   1:L PR[91] R[100]mm/sec CNT100;
   1:  PR[GP1:91,1] = PR[GP1:90,1] + -54.768;
   1:  PR[GP1:91,2] = PR[GP1:90,2] + 21.323;
   1:L PR[91] R[100]mm/sec CNT100;
   1:  PR[GP1:91,1] = PR[GP1:90,1] + -59.783;
   1:  PR[GP1:91,2] = PR[GP1:90,2] + 12.944;
   1:L PR[91] R[100]mm/sec CNT100;
   1:  PR[GP1:91,1] = PR[GP1:90,1] + -60.363;
   1:  PR[GP1:91,2] = PR[GP1:90,2] + 10.978;
   1:L PR[91] R[100]mm/sec CNT100;
   1:  PR[GP1:91,1] = PR[GP1:90,1] + -60.560;
   1:  PR[GP1:91,2] = PR[GP1:90,2] + 8.823;
   1:L PR[91] R[100]mm/sec CNT100;
   1:  PR[GP1:91,1] = PR[GP1:90,1] + -62.205;
   1:  PR[GP1:91,2] = PR[GP1:90,2] + -0.100;
   1:L PR[91] R[100]mm/sec CNT100;
   1:  PR[GP1:91,1] = PR[GP1:90,1] + -62.009;
   1:  PR[GP1:91,2] = PR[GP1:90,2] + -2.267;
   1:L PR[91] R[100]mm/sec CNT100;
   1:  PR[GP1:91,1] = PR[GP1:90,1] + -60.370;
   1:  PR[GP1:91,2] = PR[GP1:90,2] + -11.098;
   1:L PR[91] R[100]mm/sec CNT100;
   1:  PR[GP1:91,1] = PR[GP1:90,1] + -59.777;
   1:  PR[GP1:91,2] = PR[GP1:90,2] + -13.111;
   1:L PR[91] R[100]mm/sec CNT100;
   1:  PR[GP1:91,1] = PR[GP1:90,1] + -58.814;
   1:  PR[GP1:91,2] = PR[GP1:90,2] + -14.997;
   1:L PR[91] R[100]mm/sec CNT100;
   1:  PR[GP1:91,1] = PR[GP1:90,1] + -53.831;
   1:  PR[GP1:91,2] = PR[GP1:90,2] + -23.288;
   1:L PR[91] R[100]mm/sec CNT100;
   1:  PR[GP1:91,1] = PR[GP1:90,1] + -52.724;
   1:  PR[GP1:91,2] = PR[GP1:90,2] + -24.729;
   1:L PR[91] R[100]mm/sec CNT100;
   1:  PR[GP1:91,1] = PR[GP1:90,1] + -51.475;
   1:  PR[GP1:91,2] = PR[GP1:90,2] + -25.850;
   1:L PR[91] R[100]mm/sec CNT100;
   1:  PR[GP1:91,1] = PR[GP1:90,1] + -43.113;
   1:  PR[GP1:91,2] = PR[GP1:90,2] + -32.589;
   1:L PR[91] R[100]mm/sec CNT100;
   1:  PR[GP1:91,1] = PR[GP1:90,1] + -41.986;
   1:  PR[GP1:91,2] = PR[GP1:90,2] + -33.291;
   1:L PR[91] R[100]mm/sec CNT100;
   1:  PR[GP1:91,1] = PR[GP1:90,1] + -40.875;
   1:  PR[GP1:91,2] = PR[GP1:90,2] + -33.737;
   1:L PR[91] R[100]mm/sec CNT100;
   1:  PR[GP1:91,1] = PR[GP1:90,1] + -29.510;
   1:  PR[GP1:91,2] = PR[GP1:90,2] + -37.747;
   1:L PR[91] R[100]mm/sec CNT100;
   1:  PR[GP1:91,1] = PR[GP1:90,1] + -28.836;
   1:  PR[GP1:91,2] = PR[GP1:90,2] + -37.892;
   1:L PR[91] R[100]mm/sec CNT100;
   1:  PR[GP1:91,1] = PR[GP1:90,1] + -28.211;
   1:  PR[GP1:91,2] = PR[GP1:90,2] + -37.917;
   1:L PR[91] R[100]mm/sec CNT100;
   1:  PR[GP1:91,1] = PR[GP1:90,1] + -14.890;
   1:  PR[GP1:91,2] = PR[GP1:90,2] + -37.959;
   1:L PR[91] R[100]mm/sec CNT100;
   1:  PR[GP1:91,1] = PR[GP1:90,1] + -14.841;
   1:  PR[GP1:91,2] = PR[GP1:90,2] + -37.952;
   1:L PR[91] R[100]mm/sec CNT100;
   1:  PR[GP1:91,1] = PR[GP1:90,1] + -14.779;
   1:  PR[GP1:91,2] = PR[GP1:90,2] + -37.932;
   1:L PR[91] R[100]mm/sec CNT100;
   1:  PR[GP1:91,1] = PR[GP1:90,1] + -11.835;
   1:  PR[GP1:91,2] = PR[GP1:90,2] + -36.909;
   1:L PR[91] R[100]mm/sec CNT100;
   1:  PR[GP1:91,1] = PR[GP1:90,1] + -2.186;
   1:  PR[GP1:91,2] = PR[GP1:90,2] + -33.761;
   1:L PR[91] R[100]mm/sec CNT100;
   1:  PR[GP1:91,1] = PR[GP1:90,1] + -0.355;
   1:  PR[GP1:91,2] = PR[GP1:90,2] + -33.769;
   1:L PR[91] R[100]mm/sec CNT100;
   1:  PR[GP1:91,1] = PR[GP1:90,1] + 1.412;
   1:  PR[GP1:91,2] = PR[GP1:90,2] + -33.699;
   1:L PR[91] R[100]mm/sec CNT100;
   1:  PR[GP1:91,1] = PR[GP1:90,1] + 2.210;
   1:  PR[GP1:91,2] = PR[GP1:90,2] + -33.528;
   1:L PR[91] R[100]mm/sec CNT100;
   1:  PR[GP1:91,1] = PR[GP1:90,1] + 2.588;
   1:  PR[GP1:91,2] = PR[GP1:90,2] + -33.832;
   1:L PR[91] R[100]mm/sec CNT100;
   1:  PR[GP1:91,1] = PR[GP1:90,1] + 12.046;
   1:  PR[GP1:91,2] = PR[GP1:90,2] + -36.909;
   1:L PR[91] R[100]mm/sec CNT100;
   1:  PR[GP1:91,1] = PR[GP1:90,1] + 15.059;
   1:  PR[GP1:91,2] = PR[GP1:90,2] + -37.952;
   1:L PR[91] R[100]mm/sec CNT100;
   1:  PR[GP1:91,1] = PR[GP1:90,1] + 15.099;
   1:  PR[GP1:91,2] = PR[GP1:90,2] + -37.958;
   1:L PR[91] R[100]mm/sec CNT100;
   1:  PR[GP1:91,1] = PR[GP1:90,1] + 29.053;
   1:  PR[GP1:91,2] = PR[GP1:90,2] + -37.892;
   1:L PR[91] R[100]mm/sec CNT100;
   1:  PR[GP1:91,1] = PR[GP1:90,1] + 29.705;
   1:  PR[GP1:91,2] = PR[GP1:90,2] + -37.751;
   1:L PR[91] R[100]mm/sec CNT100;
   1:  PR[GP1:91,1] = PR[GP1:90,1] + 30.492;
   1:  PR[GP1:91,2] = PR[GP1:90,2] + -37.441;
   1:L PR[91] R[100]mm/sec CNT100;
   1:  PR[GP1:91,1] = PR[GP1:90,1] + 42.202;
   1:  PR[GP1:91,2] = PR[GP1:90,2] + -33.291;
   1:L PR[91] R[100]mm/sec CNT100;
   1:  PR[GP1:91,1] = PR[GP1:90,1] + 43.299;
   1:  PR[GP1:91,2] = PR[GP1:90,2] + -32.611;
   1:L PR[91] R[100]mm/sec CNT100;
   1:  PR[GP1:91,1] = PR[GP1:90,1] + 44.416;
   1:  PR[GP1:91,2] = PR[GP1:90,2] + -31.622;
   1:L PR[91] R[100]mm/sec CNT100;
   1:  PR[GP1:91,1] = PR[GP1:90,1] + 52.923;
   1:  PR[GP1:91,2] = PR[GP1:90,2] + -24.736;
   1:L PR[91] R[100]mm/sec CNT100;
   1:  PR[GP1:91,1] = PR[GP1:90,1] + 54.021;
   1:  PR[GP1:91,2] = PR[GP1:90,2] + -23.310;
   1:L PR[91] R[100]mm/sec CNT100;
   1:  PR[GP1:91,1] = PR[GP1:90,1] + 54.968;
   1:  PR[GP1:91,2] = PR[GP1:90,2] + -21.493;
   1:L PR[91] R[100]mm/sec CNT100;
   1:  PR[GP1:91,1] = PR[GP1:90,1] + 59.987;
   1:  PR[GP1:91,2] = PR[GP1:90,2] + -13.131;
   1:L PR[91] R[100]mm/sec CNT100;
   1:  PR[GP1:91,1] = PR[GP1:90,1] + 60.565;
   1:  PR[GP1:91,2] = PR[GP1:90,2] + -11.196;
   1:L PR[91] R[100]mm/sec CNT100;
   1:  PR[GP1:91,1] = PR[GP1:90,1] + 60.772;
   1:  PR[GP1:91,2] = PR[GP1:90,2] + -8.982;
   1:L PR[91] R[100]mm/sec CNT100;
   1:  PR[GP1:91,1] = PR[GP1:90,1] + 62.418;
   1:  PR[GP1:91,2] = PR[GP1:90,2] + -0.045;
   1:L PR[91] R[100]mm/sec CNT100;
   1:  PR[GP1:91,1] = PR[GP1:90,1] + 62.212;
   1:  PR[GP1:91,2] = PR[GP1:90,2] + 2.185;
   1:L PR[91] R[100]mm/sec CNT100;
   1:  PR[GP1:91,1] = PR[GP1:90,1] + 60.574;
   1:  PR[GP1:91,2] = PR[GP1:90,2] + 11.023;
   1:L PR[91] R[100]mm/sec CNT100;
   1:  PR[GP1:91,1] = PR[GP1:90,1] + 59.982;
   1:  PR[GP1:91,2] = PR[GP1:90,2] + 13.003;
   1:L PR[91] R[100]mm/sec CNT100;
   1:  PR[GP1:91,1] = PR[GP1:90,1] + 59.017;
   1:  PR[GP1:91,2] = PR[GP1:90,2] + 14.874;
   1:L PR[91] R[100]mm/sec CNT100;
   1:  PR[GP1:91,1] = PR[GP1:90,1] + 54.037;
   1:  PR[GP1:91,2] = PR[GP1:90,2] + 23.147;
   1:L PR[91] R[100]mm/sec CNT100;
   1:  PR[GP1:91,1] = PR[GP1:90,1] + 52.918;
   1:  PR[GP1:91,2] = PR[GP1:90,2] + 24.599;
   1:L PR[91] R[100]mm/sec CNT100;
   1:  PR[GP1:91,1] = PR[GP1:90,1] + 51.675;
   1:  PR[GP1:91,2] = PR[GP1:90,2] + 25.710;
   1:L PR[91] R[100]mm/sec CNT100;
   1:  PR[GP1:91,1] = PR[GP1:90,1] + 43.320;
   1:  PR[GP1:91,2] = PR[GP1:90,2] + 32.454;
   1:L PR[91] R[100]mm/sec CNT100;
   1:  PR[GP1:91,1] = PR[GP1:90,1] + 42.201;
   1:  PR[GP1:91,2] = PR[GP1:90,2] + 33.148;
   1:L PR[91] R[100]mm/sec CNT100;
   1:  PR[GP1:91,1] = PR[GP1:90,1] + 41.088;
   1:  PR[GP1:91,2] = PR[GP1:90,2] + 33.593;
   1:L PR[91] R[100]mm/sec CNT100;
   1:  PR[GP1:91,1] = PR[GP1:90,1] + 29.731;
   1:  PR[GP1:91,2] = PR[GP1:90,2] + 37.602;
   1:L PR[91] R[100]mm/sec CNT100;
   1:  PR[GP1:91,1] = PR[GP1:90,1] + 29.058;
   1:  PR[GP1:91,2] = PR[GP1:90,2] + 37.747;
   1:L PR[91] R[100]mm/sec CNT100;
   1:  PR[GP1:91,1] = PR[GP1:90,1] + 28.436;
   1:  PR[GP1:91,2] = PR[GP1:90,2] + 37.770;
   1:L PR[91] R[100]mm/sec CNT100;
   1:  PR[GP1:91,1] = PR[GP1:90,1] + 15.122;
   1:  PR[GP1:91,2] = PR[GP1:90,2] + 37.817;
   1:L PR[91] R[100]mm/sec CNT100;
   1:  PR[GP1:91,1] = PR[GP1:90,1] + 15.080;
   1:  PR[GP1:91,2] = PR[GP1:90,2] + 37.812;
   1:L PR[91] R[100]mm/sec CNT100;
   1:  PR[GP1:91,1] = PR[GP1:90,1] + 11.996;
   1:  PR[GP1:91,2] = PR[GP1:90,2] + 36.746;
   1:L PR[91] R[100]mm/sec CNT100;
   1:  PR[GP1:91,1] = PR[GP1:90,1] + 2.808;
   1:  PR[GP1:91,2] = PR[GP1:90,2] + 33.760;
   1:L PR[91] R[100]mm/sec CNT100;
   1:  PR[GP1:91,1] = PR[GP1:90,1] + 2.180;
   1:  PR[GP1:91,2] = PR[GP1:90,2] + 33.410;
   1:L PR[91] R[100]mm/sec CNT100;
   1:  ! -- Layer/Ebene 117 -- !;
   1:  PR[91] = PR[90];
   1:  PR[GP1:91,1] = PR[GP1:90,1] + 0.156;
   1:  PR[GP1:91,2] = PR[GP1:90,2] + 33.822;
   1:  PR[GP1:91,3] = PR[GP1:90,3] + 71.675;
   1:L PR[91] R[100]mm/sec CNT100;
   1:  PR[GP1:91,1] = PR[GP1:90,1] + -2.159;
   1:  PR[GP1:91,2] = PR[GP1:90,2] + 33.808;
   1:L PR[91] R[100]mm/sec CNT100;
   1:  PR[GP1:91,1] = PR[GP1:90,1] + -14.621;
   1:  PR[GP1:91,2] = PR[GP1:90,2] + 37.873;
   1:L PR[91] R[100]mm/sec CNT100;
   1:  PR[GP1:91,1] = PR[GP1:90,1] + -28.674;
   1:  PR[GP1:91,2] = PR[GP1:90,2] + 37.800;
   1:L PR[91] R[100]mm/sec CNT100;
   1:  PR[GP1:91,1] = PR[GP1:90,1] + -29.170;
   1:  PR[GP1:91,2] = PR[GP1:90,2] + 37.693;
   1:L PR[91] R[100]mm/sec CNT100;
   1:  PR[GP1:91,1] = PR[GP1:90,1] + -29.787;
   1:  PR[GP1:91,2] = PR[GP1:90,2] + 37.449;
   1:L PR[91] R[100]mm/sec CNT100;
   1:  PR[GP1:91,1] = PR[GP1:90,1] + -41.823;
   1:  PR[GP1:91,2] = PR[GP1:90,2] + 33.175;
   1:L PR[91] R[100]mm/sec CNT100;
   1:  PR[GP1:91,1] = PR[GP1:90,1] + -42.785;
   1:  PR[GP1:91,2] = PR[GP1:90,2] + 32.575;
   1:L PR[91] R[100]mm/sec CNT100;
   1:  PR[GP1:91,1] = PR[GP1:90,1] + -43.774;
   1:  PR[GP1:91,2] = PR[GP1:90,2] + 31.698;
   1:L PR[91] R[100]mm/sec CNT100;
   1:  PR[GP1:91,1] = PR[GP1:90,1] + -52.554;
   1:  PR[GP1:91,2] = PR[GP1:90,2] + 24.593;
   1:L PR[91] R[100]mm/sec CNT100;
   1:  PR[GP1:91,1] = PR[GP1:90,1] + -53.539;
   1:  PR[GP1:91,2] = PR[GP1:90,2] + 23.311;
   1:L PR[91] R[100]mm/sec CNT100;
   1:  PR[GP1:91,1] = PR[GP1:90,1] + -54.399;
   1:  PR[GP1:91,2] = PR[GP1:90,2] + 21.641;
   1:L PR[91] R[100]mm/sec CNT100;
   1:  PR[GP1:91,1] = PR[GP1:90,1] + -59.596;
   1:  PR[GP1:91,2] = PR[GP1:90,2] + 12.960;
   1:L PR[91] R[100]mm/sec CNT100;
   1:  PR[GP1:91,1] = PR[GP1:90,1] + -60.130;
   1:  PR[GP1:91,2] = PR[GP1:90,2] + 11.150;
   1:L PR[91] R[100]mm/sec CNT100;
   1:  PR[GP1:91,1] = PR[GP1:90,1] + -60.312;
   1:  PR[GP1:91,2] = PR[GP1:90,2] + 9.158;
   1:L PR[91] R[100]mm/sec CNT100;
   1:  PR[GP1:91,1] = PR[GP1:90,1] + -62.019;
   1:  PR[GP1:91,2] = PR[GP1:90,2] + -0.100;
   1:L PR[91] R[100]mm/sec CNT100;
   1:  PR[GP1:91,1] = PR[GP1:90,1] + -61.837;
   1:  PR[GP1:91,2] = PR[GP1:90,2] + -2.111;
   1:L PR[91] R[100]mm/sec CNT100;
   1:  PR[GP1:91,1] = PR[GP1:90,1] + -60.137;
   1:  PR[GP1:91,2] = PR[GP1:90,2] + -11.270;
   1:L PR[91] R[100]mm/sec CNT100;
   1:  PR[GP1:91,1] = PR[GP1:90,1] + -59.589;
   1:  PR[GP1:91,2] = PR[GP1:90,2] + -13.126;
   1:L PR[91] R[100]mm/sec CNT100;
   1:  PR[GP1:91,1] = PR[GP1:90,1] + -58.701;
   1:  PR[GP1:91,2] = PR[GP1:90,2] + -14.867;
   1:L PR[91] R[100]mm/sec CNT100;
   1:  PR[GP1:91,1] = PR[GP1:90,1] + -53.546;
   1:  PR[GP1:91,2] = PR[GP1:90,2] + -23.444;
   1:L PR[91] R[100]mm/sec CNT100;
   1:  PR[GP1:91,1] = PR[GP1:90,1] + -52.540;
   1:  PR[GP1:91,2] = PR[GP1:90,2] + -24.754;
   1:L PR[91] R[100]mm/sec CNT100;
   1:  PR[GP1:91,1] = PR[GP1:90,1] + -51.405;
   1:  PR[GP1:91,2] = PR[GP1:90,2] + -25.772;
   1:L PR[91] R[100]mm/sec CNT100;
   1:  PR[GP1:91,1] = PR[GP1:90,1] + -42.788;
   1:  PR[GP1:91,2] = PR[GP1:90,2] + -32.718;
   1:L PR[91] R[100]mm/sec CNT100;
   1:  PR[GP1:91,1] = PR[GP1:90,1] + -41.802;
   1:  PR[GP1:91,2] = PR[GP1:90,2] + -33.331;
   1:L PR[91] R[100]mm/sec CNT100;
   1:  PR[GP1:91,1] = PR[GP1:90,1] + -40.829;
   1:  PR[GP1:91,2] = PR[GP1:90,2] + -33.722;
   1:L PR[91] R[100]mm/sec CNT100;
   1:  PR[GP1:91,1] = PR[GP1:90,1] + -29.164;
   1:  PR[GP1:91,2] = PR[GP1:90,2] + -37.838;
   1:L PR[91] R[100]mm/sec CNT100;
   1:  PR[GP1:91,1] = PR[GP1:90,1] + -28.648;
   1:  PR[GP1:91,2] = PR[GP1:90,2] + -37.949;
   1:L PR[91] R[100]mm/sec CNT100;
   1:  PR[GP1:91,1] = PR[GP1:90,1] + -28.166;
   1:  PR[GP1:91,2] = PR[GP1:90,2] + -37.968;
   1:L PR[91] R[100]mm/sec CNT100;
   1:  PR[GP1:91,1] = PR[GP1:90,1] + -14.623;
   1:  PR[GP1:91,2] = PR[GP1:90,2] + -38.014;
   1:L PR[91] R[100]mm/sec CNT100;
   1:  PR[GP1:91,1] = PR[GP1:90,1] + -2.159;
   1:  PR[GP1:91,2] = PR[GP1:90,2] + -33.955;
   1:L PR[91] R[100]mm/sec CNT100;
   1:  PR[GP1:91,1] = PR[GP1:90,1] + 0.246;
   1:  PR[GP1:91,2] = PR[GP1:90,2] + -33.967;
   1:L PR[91] R[100]mm/sec CNT100;
   1:  PR[GP1:91,1] = PR[GP1:90,1] + 1.578;
   1:  PR[GP1:91,2] = PR[GP1:90,2] + -33.913;
   1:L PR[91] R[100]mm/sec CNT100;
   1:  PR[GP1:91,1] = PR[GP1:90,1] + 2.241;
   1:  PR[GP1:91,2] = PR[GP1:90,2] + -33.772;
   1:L PR[91] R[100]mm/sec CNT100;
   1:  PR[GP1:91,1] = PR[GP1:90,1] + 2.561;
   1:  PR[GP1:91,2] = PR[GP1:90,2] + -34.030;
   1:L PR[91] R[100]mm/sec CNT100;
   1:  PR[GP1:91,1] = PR[GP1:90,1] + 14.808;
   1:  PR[GP1:91,2] = PR[GP1:90,2] + -38.012;
   1:L PR[91] R[100]mm/sec CNT100;
   1:  PR[GP1:91,1] = PR[GP1:90,1] + 28.865;
   1:  PR[GP1:91,2] = PR[GP1:90,2] + -37.948;
   1:L PR[91] R[100]mm/sec CNT100;
   1:  PR[GP1:91,1] = PR[GP1:90,1] + 29.360;
   1:  PR[GP1:91,2] = PR[GP1:90,2] + -37.842;
   1:L PR[91] R[100]mm/sec CNT100;
   1:  PR[GP1:91,1] = PR[GP1:90,1] + 29.977;
   1:  PR[GP1:91,2] = PR[GP1:90,2] + -37.599;
   1:L PR[91] R[100]mm/sec CNT100;
   1:  PR[GP1:91,1] = PR[GP1:90,1] + 42.019;
   1:  PR[GP1:91,2] = PR[GP1:90,2] + -33.331;
   1:L PR[91] R[100]mm/sec CNT100;
   1:  PR[GP1:91,1] = PR[GP1:90,1] + 42.976;
   1:  PR[GP1:91,2] = PR[GP1:90,2] + -32.738;
   1:L PR[91] R[100]mm/sec CNT100;
   1:  PR[GP1:91,1] = PR[GP1:90,1] + 43.957;
   1:  PR[GP1:91,2] = PR[GP1:90,2] + -31.869;
   1:L PR[91] R[100]mm/sec CNT100;
   1:  PR[GP1:91,1] = PR[GP1:90,1] + 52.741;
   1:  PR[GP1:91,2] = PR[GP1:90,2] + -24.758;
   1:L PR[91] R[100]mm/sec CNT100;
   1:  PR[GP1:91,1] = PR[GP1:90,1] + 53.737;
   1:  PR[GP1:91,2] = PR[GP1:90,2] + -23.465;
   1:L PR[91] R[100]mm/sec CNT100;
   1:  PR[GP1:91,1] = PR[GP1:90,1] + 54.600;
   1:  PR[GP1:91,2] = PR[GP1:90,2] + -21.809;
   1:L PR[91] R[100]mm/sec CNT100;
   1:  PR[GP1:91,1] = PR[GP1:90,1] + 59.801;
   1:  PR[GP1:91,2] = PR[GP1:90,2] + -13.145;
   1:L PR[91] R[100]mm/sec CNT100;
   1:  PR[GP1:91,1] = PR[GP1:90,1] + 60.333;
   1:  PR[GP1:91,2] = PR[GP1:90,2] + -11.363;
   1:L PR[91] R[100]mm/sec CNT100;
   1:  PR[GP1:91,1] = PR[GP1:90,1] + 60.524;
   1:  PR[GP1:91,2] = PR[GP1:90,2] + -9.317;
   1:L PR[91] R[100]mm/sec CNT100;
   1:  PR[GP1:91,1] = PR[GP1:90,1] + 62.232;
   1:  PR[GP1:91,2] = PR[GP1:90,2] + -0.045;
   1:L PR[91] R[100]mm/sec CNT100;
   1:  PR[GP1:91,1] = PR[GP1:90,1] + 62.041;
   1:  PR[GP1:91,2] = PR[GP1:90,2] + 2.024;
   1:L PR[91] R[100]mm/sec CNT100;
   1:  PR[GP1:91,1] = PR[GP1:90,1] + 60.342;
   1:  PR[GP1:91,2] = PR[GP1:90,2] + 11.191;
   1:L PR[91] R[100]mm/sec CNT100;
   1:  PR[GP1:91,1] = PR[GP1:90,1] + 59.796;
   1:  PR[GP1:91,2] = PR[GP1:90,2] + 13.017;
   1:L PR[91] R[100]mm/sec CNT100;
   1:  PR[GP1:91,1] = PR[GP1:90,1] + 58.905;
   1:  PR[GP1:91,2] = PR[GP1:90,2] + 14.743;
   1:L PR[91] R[100]mm/sec CNT100;
   1:  PR[GP1:91,1] = PR[GP1:90,1] + 53.753;
   1:  PR[GP1:91,2] = PR[GP1:90,2] + 23.301;
   1:L PR[91] R[100]mm/sec CNT100;
   1:  PR[GP1:91,1] = PR[GP1:90,1] + 52.737;
   1:  PR[GP1:91,2] = PR[GP1:90,2] + 24.621;
   1:L PR[91] R[100]mm/sec CNT100;
   1:  PR[GP1:91,1] = PR[GP1:90,1] + 51.607;
   1:  PR[GP1:91,2] = PR[GP1:90,2] + 25.631;
   1:L PR[91] R[100]mm/sec CNT100;
   1:  PR[GP1:91,1] = PR[GP1:90,1] + 42.997;
   1:  PR[GP1:91,2] = PR[GP1:90,2] + 32.581;
   1:L PR[91] R[100]mm/sec CNT100;
   1:  PR[GP1:91,1] = PR[GP1:90,1] + 42.019;
   1:  PR[GP1:91,2] = PR[GP1:90,2] + 33.188;
   1:L PR[91] R[100]mm/sec CNT100;
   1:  PR[GP1:91,1] = PR[GP1:90,1] + 41.044;
   1:  PR[GP1:91,2] = PR[GP1:90,2] + 33.577;
   1:L PR[91] R[100]mm/sec CNT100;
   1:  PR[GP1:91,1] = PR[GP1:90,1] + 29.387;
   1:  PR[GP1:91,2] = PR[GP1:90,2] + 37.693;
   1:L PR[91] R[100]mm/sec CNT100;
   1:  PR[GP1:91,1] = PR[GP1:90,1] + 28.871;
   1:  PR[GP1:91,2] = PR[GP1:90,2] + 37.803;
   1:L PR[91] R[100]mm/sec CNT100;
   1:  PR[GP1:91,1] = PR[GP1:90,1] + 28.391;
   1:  PR[GP1:91,2] = PR[GP1:90,2] + 37.822;
   1:L PR[91] R[100]mm/sec CNT100;
   1:  PR[GP1:91,1] = PR[GP1:90,1] + 14.829;
   1:  PR[GP1:91,2] = PR[GP1:90,2] + 37.872;
   1:L PR[91] R[100]mm/sec CNT100;
   1:  PR[GP1:91,1] = PR[GP1:90,1] + 2.720;
   1:  PR[GP1:91,2] = PR[GP1:90,2] + 33.937;
   1:L PR[91] R[100]mm/sec CNT100;
   1:  PR[GP1:91,1] = PR[GP1:90,1] + 2.210;
   1:  PR[GP1:91,2] = PR[GP1:90,2] + 33.653;
   1:L PR[91] R[100]mm/sec CNT100;
   1:  ! -- Layer/Ebene 118 -- !;
   1:  PR[91] = PR[90];
   1:  PR[GP1:91,1] = PR[GP1:90,1] + 0.747;
   1:  PR[GP1:91,2] = PR[GP1:90,2] + 34.019;
   1:  PR[GP1:91,3] = PR[GP1:90,3] + 72.285;
   1:L PR[91] R[100]mm/sec CNT100;
   1:  PR[GP1:91,1] = PR[GP1:90,1] + -2.132;
   1:  PR[GP1:91,2] = PR[GP1:90,2] + 34.002;
   1:L PR[91] R[100]mm/sec CNT100;
   1:  PR[GP1:91,1] = PR[GP1:90,1] + -13.373;
   1:  PR[GP1:91,2] = PR[GP1:90,2] + 37.669;
   1:L PR[91] R[100]mm/sec CNT100;
   1:  PR[GP1:91,1] = PR[GP1:90,1] + -14.331;
   1:  PR[GP1:91,2] = PR[GP1:90,2] + 37.965;
   1:L PR[91] R[100]mm/sec CNT100;
   1:  PR[GP1:91,1] = PR[GP1:90,1] + -14.593;
   1:  PR[GP1:91,2] = PR[GP1:90,2] + 37.974;
   1:L PR[91] R[100]mm/sec CNT100;
   1:  PR[GP1:91,1] = PR[GP1:90,1] + -18.226;
   1:  PR[GP1:91,2] = PR[GP1:90,2] + 37.908;
   1:L PR[91] R[100]mm/sec CNT100;
   1:  PR[GP1:91,1] = PR[GP1:90,1] + -28.487;
   1:  PR[GP1:91,2] = PR[GP1:90,2] + 37.857;
   1:L PR[91] R[100]mm/sec CNT100;
   1:  PR[GP1:91,1] = PR[GP1:90,1] + -28.825;
   1:  PR[GP1:91,2] = PR[GP1:90,2] + 37.784;
   1:L PR[91] R[100]mm/sec CNT100;
   1:  PR[GP1:91,1] = PR[GP1:90,1] + -29.271;
   1:  PR[GP1:91,2] = PR[GP1:90,2] + 37.607;
   1:L PR[91] R[100]mm/sec CNT100;
   1:  PR[GP1:91,1] = PR[GP1:90,1] + -41.639;
   1:  PR[GP1:91,2] = PR[GP1:90,2] + 33.215;
   1:L PR[91] R[100]mm/sec CNT100;
   1:  PR[GP1:91,1] = PR[GP1:90,1] + -42.461;
   1:  PR[GP1:91,2] = PR[GP1:90,2] + 32.704;
   1:L PR[91] R[100]mm/sec CNT100;
   1:  PR[GP1:91,1] = PR[GP1:90,1] + -43.313;
   1:  PR[GP1:91,2] = PR[GP1:90,2] + 31.946;
   1:L PR[91] R[100]mm/sec CNT100;
   1:  PR[GP1:91,1] = PR[GP1:90,1] + -52.371;
   1:  PR[GP1:91,2] = PR[GP1:90,2] + 24.617;
   1:L PR[91] R[100]mm/sec CNT100;
   1:  PR[GP1:91,1] = PR[GP1:90,1] + -53.254;
   1:  PR[GP1:91,2] = PR[GP1:90,2] + 23.467;
   1:L PR[91] R[100]mm/sec CNT100;
   1:  PR[GP1:91,1] = PR[GP1:90,1] + -54.031;
   1:  PR[GP1:91,2] = PR[GP1:90,2] + 21.959;
   1:L PR[91] R[100]mm/sec CNT100;
   1:  PR[GP1:91,1] = PR[GP1:90,1] + -59.409;
   1:  PR[GP1:91,2] = PR[GP1:90,2] + 12.975;
   1:L PR[91] R[100]mm/sec CNT100;
   1:  PR[GP1:91,1] = PR[GP1:90,1] + -59.897;
   1:  PR[GP1:91,2] = PR[GP1:90,2] + 11.321;
   1:L PR[91] R[100]mm/sec CNT100;
   1:  PR[GP1:91,1] = PR[GP1:90,1] + -60.064;
   1:  PR[GP1:91,2] = PR[GP1:90,2] + 9.492;
   1:L PR[91] R[100]mm/sec CNT100;
   1:  PR[GP1:91,1] = PR[GP1:90,1] + -61.832;
   1:  PR[GP1:91,2] = PR[GP1:90,2] + -0.100;
   1:L PR[91] R[100]mm/sec CNT100;
   1:  PR[GP1:91,1] = PR[GP1:90,1] + -61.665;
   1:  PR[GP1:91,2] = PR[GP1:90,2] + -1.954;
   1:L PR[91] R[100]mm/sec CNT100;
   1:  PR[GP1:91,1] = PR[GP1:90,1] + -59.903;
   1:  PR[GP1:91,2] = PR[GP1:90,2] + -11.442;
   1:L PR[91] R[100]mm/sec CNT100;
   1:  PR[GP1:91,1] = PR[GP1:90,1] + -59.402;
   1:  PR[GP1:91,2] = PR[GP1:90,2] + -13.142;
   1:L PR[91] R[100]mm/sec CNT100;
   1:  PR[GP1:91,1] = PR[GP1:90,1] + -58.589;
   1:  PR[GP1:91,2] = PR[GP1:90,2] + -14.737;
   1:L PR[91] R[100]mm/sec CNT100;
   1:  PR[GP1:91,1] = PR[GP1:90,1] + -53.262;
   1:  PR[GP1:91,2] = PR[GP1:90,2] + -23.600;
   1:L PR[91] R[100]mm/sec CNT100;
   1:  PR[GP1:91,1] = PR[GP1:90,1] + -52.357;
   1:  PR[GP1:91,2] = PR[GP1:90,2] + -24.778;
   1:L PR[91] R[100]mm/sec CNT100;
   1:  PR[GP1:91,1] = PR[GP1:90,1] + -51.334;
   1:  PR[GP1:91,2] = PR[GP1:90,2] + -25.695;
   1:L PR[91] R[100]mm/sec CNT100;
   1:  PR[GP1:91,1] = PR[GP1:90,1] + -42.462;
   1:  PR[GP1:91,2] = PR[GP1:90,2] + -32.846;
   1:L PR[91] R[100]mm/sec CNT100;
   1:  PR[GP1:91,1] = PR[GP1:90,1] + -41.619;
   1:  PR[GP1:91,2] = PR[GP1:90,2] + -33.371;
   1:L PR[91] R[100]mm/sec CNT100;
   1:  PR[GP1:91,1] = PR[GP1:90,1] + -40.783;
   1:  PR[GP1:91,2] = PR[GP1:90,2] + -33.707;
   1:L PR[91] R[100]mm/sec CNT100;
   1:  PR[GP1:91,1] = PR[GP1:90,1] + -28.818;
   1:  PR[GP1:91,2] = PR[GP1:90,2] + -37.928;
   1:L PR[91] R[100]mm/sec CNT100;
   1:  PR[GP1:91,1] = PR[GP1:90,1] + -28.460;
   1:  PR[GP1:91,2] = PR[GP1:90,2] + -38.006;
   1:L PR[91] R[100]mm/sec CNT100;
   1:  PR[GP1:91,1] = PR[GP1:90,1] + -28.120;
   1:  PR[GP1:91,2] = PR[GP1:90,2] + -38.019;
   1:L PR[91] R[100]mm/sec CNT100;
   1:  PR[GP1:91,1] = PR[GP1:90,1] + -18.226;
   1:  PR[GP1:91,2] = PR[GP1:90,2] + -38.050;
   1:L PR[91] R[100]mm/sec CNT100;
   1:  PR[GP1:91,1] = PR[GP1:90,1] + -14.573;
   1:  PR[GP1:91,2] = PR[GP1:90,2] + -38.115;
   1:L PR[91] R[100]mm/sec CNT100;
   1:  PR[GP1:91,1] = PR[GP1:90,1] + -14.309;
   1:  PR[GP1:91,2] = PR[GP1:90,2] + -38.106;
   1:L PR[91] R[100]mm/sec CNT100;
   1:  PR[GP1:91,1] = PR[GP1:90,1] + -13.125;
   1:  PR[GP1:91,2] = PR[GP1:90,2] + -37.737;
   1:L PR[91] R[100]mm/sec CNT100;
   1:  PR[GP1:91,1] = PR[GP1:90,1] + -2.132;
   1:  PR[GP1:91,2] = PR[GP1:90,2] + -34.149;
   1:L PR[91] R[100]mm/sec CNT100;
   1:  PR[GP1:91,1] = PR[GP1:90,1] + 0.848;
   1:  PR[GP1:91,2] = PR[GP1:90,2] + -34.164;
   1:L PR[91] R[100]mm/sec CNT100;
   1:  PR[GP1:91,1] = PR[GP1:90,1] + 1.743;
   1:  PR[GP1:91,2] = PR[GP1:90,2] + -34.128;
   1:L PR[91] R[100]mm/sec CNT100;
   1:  PR[GP1:91,1] = PR[GP1:90,1] + 2.271;
   1:  PR[GP1:91,2] = PR[GP1:90,2] + -34.016;
   1:L PR[91] R[100]mm/sec CNT100;
   1:  PR[GP1:91,1] = PR[GP1:90,1] + 2.534;
   1:  PR[GP1:91,2] = PR[GP1:90,2] + -34.227;
   1:L PR[91] R[100]mm/sec CNT100;
   1:  PR[GP1:91,1] = PR[GP1:90,1] + 10.808;
   1:  PR[GP1:91,2] = PR[GP1:90,2] + -36.919;
   1:L PR[91] R[100]mm/sec CNT100;
   1:  PR[GP1:91,1] = PR[GP1:90,1] + 14.521;
   1:  PR[GP1:91,2] = PR[GP1:90,2] + -38.105;
   1:L PR[91] R[100]mm/sec CNT100;
   1:  PR[GP1:91,1] = PR[GP1:90,1] + 14.783;
   1:  PR[GP1:91,2] = PR[GP1:90,2] + -38.114;
   1:L PR[91] R[100]mm/sec CNT100;
   1:  PR[GP1:91,1] = PR[GP1:90,1] + 18.439;
   1:  PR[GP1:91,2] = PR[GP1:90,2] + -38.050;
   1:L PR[91] R[100]mm/sec CNT100;
   1:  PR[GP1:91,1] = PR[GP1:90,1] + 28.678;
   1:  PR[GP1:91,2] = PR[GP1:90,2] + -38.005;
   1:L PR[91] R[100]mm/sec CNT100;
   1:  PR[GP1:91,1] = PR[GP1:90,1] + 29.015;
   1:  PR[GP1:91,2] = PR[GP1:90,2] + -37.932;
   1:L PR[91] R[100]mm/sec CNT100;
   1:  PR[GP1:91,1] = PR[GP1:90,1] + 29.461;
   1:  PR[GP1:91,2] = PR[GP1:90,2] + -37.756;
   1:L PR[91] R[100]mm/sec CNT100;
   1:  PR[GP1:91,1] = PR[GP1:90,1] + 41.836;
   1:  PR[GP1:91,2] = PR[GP1:90,2] + -33.370;
   1:L PR[91] R[100]mm/sec CNT100;
   1:  PR[GP1:91,1] = PR[GP1:90,1] + 42.652;
   1:  PR[GP1:91,2] = PR[GP1:90,2] + -32.865;
   1:L PR[91] R[100]mm/sec CNT100;
   1:  PR[GP1:91,1] = PR[GP1:90,1] + 43.499;
   1:  PR[GP1:91,2] = PR[GP1:90,2] + -32.115;
   1:L PR[91] R[100]mm/sec CNT100;
   1:  PR[GP1:91,1] = PR[GP1:90,1] + 52.560;
   1:  PR[GP1:91,2] = PR[GP1:90,2] + -24.780;
   1:L PR[91] R[100]mm/sec CNT100;
   1:  PR[GP1:91,1] = PR[GP1:90,1] + 53.454;
   1:  PR[GP1:91,2] = PR[GP1:90,2] + -23.620;
   1:L PR[91] R[100]mm/sec CNT100;
   1:  PR[GP1:91,1] = PR[GP1:90,1] + 54.233;
   1:  PR[GP1:91,2] = PR[GP1:90,2] + -22.125;
   1:L PR[91] R[100]mm/sec CNT100;
   1:  PR[GP1:91,1] = PR[GP1:90,1] + 59.614;
   1:  PR[GP1:91,2] = PR[GP1:90,2] + -13.159;
   1:L PR[91] R[100]mm/sec CNT100;
   1:  PR[GP1:91,1] = PR[GP1:90,1] + 60.101;
   1:  PR[GP1:91,2] = PR[GP1:90,2] + -11.531;
   1:L PR[91] R[100]mm/sec CNT100;
   1:  PR[GP1:91,1] = PR[GP1:90,1] + 60.276;
   1:  PR[GP1:91,2] = PR[GP1:90,2] + -9.651;
   1:L PR[91] R[100]mm/sec CNT100;
   1:  PR[GP1:91,1] = PR[GP1:90,1] + 62.045;
   1:  PR[GP1:91,2] = PR[GP1:90,2] + -0.045;
   1:L PR[91] R[100]mm/sec CNT100;
   1:  PR[GP1:91,1] = PR[GP1:90,1] + 61.869;
   1:  PR[GP1:91,2] = PR[GP1:90,2] + 1.863;
   1:L PR[91] R[100]mm/sec CNT100;
   1:  PR[GP1:91,1] = PR[GP1:90,1] + 60.109;
   1:  PR[GP1:91,2] = PR[GP1:90,2] + 11.358;
   1:L PR[91] R[100]mm/sec CNT100;
   1:  PR[GP1:91,1] = PR[GP1:90,1] + 59.610;
   1:  PR[GP1:91,2] = PR[GP1:90,2] + 13.031;
   1:L PR[91] R[100]mm/sec CNT100;
   1:  PR[GP1:91,1] = PR[GP1:90,1] + 58.793;
   1:  PR[GP1:91,2] = PR[GP1:90,2] + 14.613;
   1:L PR[91] R[100]mm/sec CNT100;
   1:  PR[GP1:91,1] = PR[GP1:90,1] + 53.469;
   1:  PR[GP1:91,2] = PR[GP1:90,2] + 23.456;
   1:L PR[91] R[100]mm/sec CNT100;
   1:  PR[GP1:91,1] = PR[GP1:90,1] + 52.555;
   1:  PR[GP1:91,2] = PR[GP1:90,2] + 24.643;
   1:L PR[91] R[100]mm/sec CNT100;
   1:  PR[GP1:91,1] = PR[GP1:90,1] + 51.538;
   1:  PR[GP1:91,2] = PR[GP1:90,2] + 25.552;
   1:L PR[91] R[100]mm/sec CNT100;
   1:  PR[GP1:91,1] = PR[GP1:90,1] + 42.674;
   1:  PR[GP1:91,2] = PR[GP1:90,2] + 32.708;
   1:L PR[91] R[100]mm/sec CNT100;
   1:  PR[GP1:91,1] = PR[GP1:90,1] + 41.836;
   1:  PR[GP1:91,2] = PR[GP1:90,2] + 33.227;
   1:L PR[91] R[100]mm/sec CNT100;
   1:  PR[GP1:91,1] = PR[GP1:90,1] + 40.999;
   1:  PR[GP1:91,2] = PR[GP1:90,2] + 33.562;
   1:L PR[91] R[100]mm/sec CNT100;
   1:  PR[GP1:91,1] = PR[GP1:90,1] + 29.042;
   1:  PR[GP1:91,2] = PR[GP1:90,2] + 37.783;
   1:L PR[91] R[100]mm/sec CNT100;
   1:  PR[GP1:91,1] = PR[GP1:90,1] + 28.685;
   1:  PR[GP1:91,2] = PR[GP1:90,2] + 37.860;
   1:L PR[91] R[100]mm/sec CNT100;
   1:  PR[GP1:91,1] = PR[GP1:90,1] + 28.346;
   1:  PR[GP1:91,2] = PR[GP1:90,2] + 37.873;
   1:L PR[91] R[100]mm/sec CNT100;
   1:  PR[GP1:91,1] = PR[GP1:90,1] + 18.439;
   1:  PR[GP1:91,2] = PR[GP1:90,2] + 37.907;
   1:L PR[91] R[100]mm/sec CNT100;
   1:  PR[GP1:91,1] = PR[GP1:90,1] + 14.803;
   1:  PR[GP1:91,2] = PR[GP1:90,2] + 37.973;
   1:L PR[91] R[100]mm/sec CNT100;
   1:  PR[GP1:91,1] = PR[GP1:90,1] + 14.542;
   1:  PR[GP1:91,2] = PR[GP1:90,2] + 37.964;
   1:L PR[91] R[100]mm/sec CNT100;
   1:  PR[GP1:91,1] = PR[GP1:90,1] + 11.048;
   1:  PR[GP1:91,2] = PR[GP1:90,2] + 36.850;
   1:L PR[91] R[100]mm/sec CNT100;
   1:  PR[GP1:91,1] = PR[GP1:90,1] + 2.631;
   1:  PR[GP1:91,2] = PR[GP1:90,2] + 34.114;
   1:L PR[91] R[100]mm/sec CNT100;
   1:  PR[GP1:91,1] = PR[GP1:90,1] + 2.240;
   1:  PR[GP1:91,2] = PR[GP1:90,2] + 33.897;
   1:L PR[91] R[100]mm/sec CNT100;
   1:  ! -- Layer/Ebene 119 -- !;
   1:  PR[91] = PR[90];
   1:  PR[GP1:91,1] = PR[GP1:90,1] + 1.338;
   1:  PR[GP1:91,2] = PR[GP1:90,2] + 34.217;
   1:  PR[GP1:91,3] = PR[GP1:90,3] + 72.895;
   1:L PR[91] R[100]mm/sec CNT100;
   1:  PR[GP1:91,1] = PR[GP1:90,1] + -2.105;
   1:  PR[GP1:91,2] = PR[GP1:90,2] + 34.195;
   1:L PR[91] R[100]mm/sec CNT100;
   1:  PR[GP1:91,1] = PR[GP1:90,1] + -12.103;
   1:  PR[GP1:91,2] = PR[GP1:90,2] + 37.457;
   1:L PR[91] R[100]mm/sec CNT100;
   1:  PR[GP1:91,1] = PR[GP1:90,1] + -14.033;
   1:  PR[GP1:91,2] = PR[GP1:90,2] + 38.054;
   1:L PR[91] R[100]mm/sec CNT100;
   1:  PR[GP1:91,1] = PR[GP1:90,1] + -14.631;
   1:  PR[GP1:91,2] = PR[GP1:90,2] + 38.075;
   1:L PR[91] R[100]mm/sec CNT100;
   1:  PR[GP1:91,1] = PR[GP1:90,1] + -21.679;
   1:  PR[GP1:91,2] = PR[GP1:90,2] + 37.946;
   1:L PR[91] R[100]mm/sec CNT100;
   1:  PR[GP1:91,1] = PR[GP1:90,1] + -28.299;
   1:  PR[GP1:91,2] = PR[GP1:90,2] + 37.913;
   1:L PR[91] R[100]mm/sec CNT100;
   1:  PR[GP1:91,1] = PR[GP1:90,1] + -28.479;
   1:  PR[GP1:91,2] = PR[GP1:90,2] + 37.874;
   1:L PR[91] R[100]mm/sec CNT100;
   1:  PR[GP1:91,1] = PR[GP1:90,1] + -28.755;
   1:  PR[GP1:91,2] = PR[GP1:90,2] + 37.765;
   1:L PR[91] R[100]mm/sec CNT100;
   1:  PR[GP1:91,1] = PR[GP1:90,1] + -41.456;
   1:  PR[GP1:91,2] = PR[GP1:90,2] + 33.255;
   1:L PR[91] R[100]mm/sec CNT100;
   1:  PR[GP1:91,1] = PR[GP1:90,1] + -42.136;
   1:  PR[GP1:91,2] = PR[GP1:90,2] + 32.832;
   1:L PR[91] R[100]mm/sec CNT100;
   1:  PR[GP1:91,1] = PR[GP1:90,1] + -42.853;
   1:  PR[GP1:91,2] = PR[GP1:90,2] + 32.195;
   1:L PR[91] R[100]mm/sec CNT100;
   1:  PR[GP1:91,1] = PR[GP1:90,1] + -52.187;
   1:  PR[GP1:91,2] = PR[GP1:90,2] + 24.641;
   1:L PR[91] R[100]mm/sec CNT100;
   1:  PR[GP1:91,1] = PR[GP1:90,1] + -52.970;
   1:  PR[GP1:91,2] = PR[GP1:90,2] + 23.623;
   1:L PR[91] R[100]mm/sec CNT100;
   1:  PR[GP1:91,1] = PR[GP1:90,1] + -53.663;
   1:  PR[GP1:91,2] = PR[GP1:90,2] + 22.277;
   1:L PR[91] R[100]mm/sec CNT100;
   1:  PR[GP1:91,1] = PR[GP1:90,1] + -59.222;
   1:  PR[GP1:91,2] = PR[GP1:90,2] + 12.991;
   1:L PR[91] R[100]mm/sec CNT100;
   1:  PR[GP1:91,1] = PR[GP1:90,1] + -59.664;
   1:  PR[GP1:91,2] = PR[GP1:90,2] + 11.493;
   1:L PR[91] R[100]mm/sec CNT100;
   1:  PR[GP1:91,1] = PR[GP1:90,1] + -59.816;
   1:  PR[GP1:91,2] = PR[GP1:90,2] + 9.826;
   1:L PR[91] R[100]mm/sec CNT100;
   1:  PR[GP1:91,1] = PR[GP1:90,1] + -61.646;
   1:  PR[GP1:91,2] = PR[GP1:90,2] + -0.100;
   1:L PR[91] R[100]mm/sec CNT100;
   1:  PR[GP1:91,1] = PR[GP1:90,1] + -61.493;
   1:  PR[GP1:91,2] = PR[GP1:90,2] + -1.798;
   1:L PR[91] R[100]mm/sec CNT100;
   1:  PR[GP1:91,1] = PR[GP1:90,1] + -59.670;
   1:  PR[GP1:91,2] = PR[GP1:90,2] + -11.613;
   1:L PR[91] R[100]mm/sec CNT100;
   1:  PR[GP1:91,1] = PR[GP1:90,1] + -59.215;
   1:  PR[GP1:91,2] = PR[GP1:90,2] + -13.158;
   1:L PR[91] R[100]mm/sec CNT100;
   1:  PR[GP1:91,1] = PR[GP1:90,1] + -58.476;
   1:  PR[GP1:91,2] = PR[GP1:90,2] + -14.608;
   1:L PR[91] R[100]mm/sec CNT100;
   1:  PR[GP1:91,1] = PR[GP1:90,1] + -52.977;
   1:  PR[GP1:91,2] = PR[GP1:90,2] + -23.756;
   1:L PR[91] R[100]mm/sec CNT100;
   1:  PR[GP1:91,1] = PR[GP1:90,1] + -52.173;
   1:  PR[GP1:91,2] = PR[GP1:90,2] + -24.803;
   1:L PR[91] R[100]mm/sec CNT100;
   1:  PR[GP1:91,1] = PR[GP1:90,1] + -51.264;
   1:  PR[GP1:91,2] = PR[GP1:90,2] + -25.618;
   1:L PR[91] R[100]mm/sec CNT100;
   1:  PR[GP1:91,1] = PR[GP1:90,1] + -42.137;
   1:  PR[GP1:91,2] = PR[GP1:90,2] + -32.974;
   1:L PR[91] R[100]mm/sec CNT100;
   1:  PR[GP1:91,1] = PR[GP1:90,1] + -41.435;
   1:  PR[GP1:91,2] = PR[GP1:90,2] + -33.412;
   1:L PR[91] R[100]mm/sec CNT100;
   1:  PR[GP1:91,1] = PR[GP1:90,1] + -40.738;
   1:  PR[GP1:91,2] = PR[GP1:90,2] + -33.692;
   1:L PR[91] R[100]mm/sec CNT100;
   1:  PR[GP1:91,1] = PR[GP1:90,1] + -28.472;
   1:  PR[GP1:91,2] = PR[GP1:90,2] + -38.019;
   1:L PR[91] R[100]mm/sec CNT100;
   1:  PR[GP1:91,1] = PR[GP1:90,1] + -28.272;
   1:  PR[GP1:91,2] = PR[GP1:90,2] + -38.062;
   1:L PR[91] R[100]mm/sec CNT100;
   1:  PR[GP1:91,1] = PR[GP1:90,1] + -28.074;
   1:  PR[GP1:91,2] = PR[GP1:90,2] + -38.070;
   1:L PR[91] R[100]mm/sec CNT100;
   1:  PR[GP1:91,1] = PR[GP1:90,1] + -21.680;
   1:  PR[GP1:91,2] = PR[GP1:90,2] + -38.090;
   1:L PR[91] R[100]mm/sec CNT100;
   1:  PR[GP1:91,1] = PR[GP1:90,1] + -14.612;
   1:  PR[GP1:91,2] = PR[GP1:90,2] + -38.216;
   1:L PR[91] R[100]mm/sec CNT100;
   1:  PR[GP1:91,1] = PR[GP1:90,1] + -14.012;
   1:  PR[GP1:91,2] = PR[GP1:90,2] + -38.194;
   1:L PR[91] R[100]mm/sec CNT100;
   1:  PR[GP1:91,1] = PR[GP1:90,1] + -11.649;
   1:  PR[GP1:91,2] = PR[GP1:90,2] + -37.459;
   1:L PR[91] R[100]mm/sec CNT100;
   1:  PR[GP1:91,1] = PR[GP1:90,1] + -2.105;
   1:  PR[GP1:91,2] = PR[GP1:90,2] + -34.344;
   1:L PR[91] R[100]mm/sec CNT100;
   1:  PR[GP1:91,1] = PR[GP1:90,1] + 1.449;
   1:  PR[GP1:91,2] = PR[GP1:90,2] + -34.361;
   1:L PR[91] R[100]mm/sec CNT100;
   1:  PR[GP1:91,1] = PR[GP1:90,1] + 1.909;
   1:  PR[GP1:91,2] = PR[GP1:90,2] + -34.343;
   1:L PR[91] R[100]mm/sec CNT100;
   1:  PR[GP1:91,1] = PR[GP1:90,1] + 2.301;
   1:  PR[GP1:91,2] = PR[GP1:90,2] + -34.259;
   1:L PR[91] R[100]mm/sec CNT100;
   1:  PR[GP1:91,1] = PR[GP1:90,1] + 2.507;
   1:  PR[GP1:91,2] = PR[GP1:90,2] + -34.425;
   1:L PR[91] R[100]mm/sec CNT100;
   1:  PR[GP1:91,1] = PR[GP1:90,1] + 6.979;
   1:  PR[GP1:91,2] = PR[GP1:90,2] + -35.880;
   1:L PR[91] R[100]mm/sec CNT100;
   1:  PR[GP1:91,1] = PR[GP1:90,1] + 11.856;
   1:  PR[GP1:91,2] = PR[GP1:90,2] + -37.457;
   1:L PR[91] R[100]mm/sec CNT100;
   1:  PR[GP1:91,1] = PR[GP1:90,1] + 14.222;
   1:  PR[GP1:91,2] = PR[GP1:90,2] + -38.193;
   1:L PR[91] R[100]mm/sec CNT100;
   1:  PR[GP1:91,1] = PR[GP1:90,1] + 14.822;
   1:  PR[GP1:91,2] = PR[GP1:90,2] + -38.215;
   1:L PR[91] R[100]mm/sec CNT100;
   1:  PR[GP1:91,1] = PR[GP1:90,1] + 21.892;
   1:  PR[GP1:91,2] = PR[GP1:90,2] + -38.090;
   1:L PR[91] R[100]mm/sec CNT100;
   1:  PR[GP1:91,1] = PR[GP1:90,1] + 28.491;
   1:  PR[GP1:91,2] = PR[GP1:90,2] + -38.061;
   1:L PR[91] R[100]mm/sec CNT100;
   1:  PR[GP1:91,1] = PR[GP1:90,1] + 28.670;
   1:  PR[GP1:91,2] = PR[GP1:90,2] + -38.023;
   1:L PR[91] R[100]mm/sec CNT100;
   1:  PR[GP1:91,1] = PR[GP1:90,1] + 28.946;
   1:  PR[GP1:91,2] = PR[GP1:90,2] + -37.914;
   1:L PR[91] R[100]mm/sec CNT100;
   1:  PR[GP1:91,1] = PR[GP1:90,1] + 41.654;
   1:  PR[GP1:91,2] = PR[GP1:90,2] + -33.410;
   1:L PR[91] R[100]mm/sec CNT100;
   1:  PR[GP1:91,1] = PR[GP1:90,1] + 42.328;
   1:  PR[GP1:91,2] = PR[GP1:90,2] + -32.992;
   1:L PR[91] R[100]mm/sec CNT100;
   1:  PR[GP1:91,1] = PR[GP1:90,1] + 43.041;
   1:  PR[GP1:91,2] = PR[GP1:90,2] + -32.361;
   1:L PR[91] R[100]mm/sec CNT100;
   1:  PR[GP1:91,1] = PR[GP1:90,1] + 52.378;
   1:  PR[GP1:91,2] = PR[GP1:90,2] + -24.803;
   1:L PR[91] R[100]mm/sec CNT100;
   1:  PR[GP1:91,1] = PR[GP1:90,1] + 53.170;
   1:  PR[GP1:91,2] = PR[GP1:90,2] + -23.775;
   1:L PR[91] R[100]mm/sec CNT100;
   1:  PR[GP1:91,1] = PR[GP1:90,1] + 53.865;
   1:  PR[GP1:91,2] = PR[GP1:90,2] + -22.441;
   1:L PR[91] R[100]mm/sec CNT100;
   1:  PR[GP1:91,1] = PR[GP1:90,1] + 59.428;
   1:  PR[GP1:91,2] = PR[GP1:90,2] + -13.173;
   1:L PR[91] R[100]mm/sec CNT100;
   1:  PR[GP1:91,1] = PR[GP1:90,1] + 59.868;
   1:  PR[GP1:91,2] = PR[GP1:90,2] + -11.699;
   1:L PR[91] R[100]mm/sec CNT100;
   1:  PR[GP1:91,1] = PR[GP1:90,1] + 60.028;
   1:  PR[GP1:91,2] = PR[GP1:90,2] + -9.986;
   1:L PR[91] R[100]mm/sec CNT100;
   1:  PR[GP1:91,1] = PR[GP1:90,1] + 61.859;
   1:  PR[GP1:91,2] = PR[GP1:90,2] + -0.045;
   1:L PR[91] R[100]mm/sec CNT100;
   1:  PR[GP1:91,1] = PR[GP1:90,1] + 61.698;
   1:  PR[GP1:91,2] = PR[GP1:90,2] + 1.702;
   1:L PR[91] R[100]mm/sec CNT100;
   1:  PR[GP1:91,1] = PR[GP1:90,1] + 59.877;
   1:  PR[GP1:91,2] = PR[GP1:90,2] + 11.526;
   1:L PR[91] R[100]mm/sec CNT100;
   1:  PR[GP1:91,1] = PR[GP1:90,1] + 59.423;
   1:  PR[GP1:91,2] = PR[GP1:90,2] + 13.045;
   1:L PR[91] R[100]mm/sec CNT100;
   1:  PR[GP1:91,1] = PR[GP1:90,1] + 58.681;
   1:  PR[GP1:91,2] = PR[GP1:90,2] + 14.483;
   1:L PR[91] R[100]mm/sec CNT100;
   1:  PR[GP1:91,1] = PR[GP1:90,1] + 53.186;
   1:  PR[GP1:91,2] = PR[GP1:90,2] + 23.611;
   1:L PR[91] R[100]mm/sec CNT100;
   1:  PR[GP1:91,1] = PR[GP1:90,1] + 52.374;
   1:  PR[GP1:91,2] = PR[GP1:90,2] + 24.665;
   1:L PR[91] R[100]mm/sec CNT100;
   1:  PR[GP1:91,1] = PR[GP1:90,1] + 51.469;
   1:  PR[GP1:91,2] = PR[GP1:90,2] + 25.474;
   1:L PR[91] R[100]mm/sec CNT100;
   1:  PR[GP1:91,1] = PR[GP1:90,1] + 42.350;
   1:  PR[GP1:91,2] = PR[GP1:90,2] + 32.835;
   1:L PR[91] R[100]mm/sec CNT100;
   1:  PR[GP1:91,1] = PR[GP1:90,1] + 41.653;
   1:  PR[GP1:91,2] = PR[GP1:90,2] + 33.267;
   1:L PR[91] R[100]mm/sec CNT100;
   1:  PR[GP1:91,1] = PR[GP1:90,1] + 40.954;
   1:  PR[GP1:91,2] = PR[GP1:90,2] + 33.546;
   1:L PR[91] R[100]mm/sec CNT100;
   1:  PR[GP1:91,1] = PR[GP1:90,1] + 28.698;
   1:  PR[GP1:91,2] = PR[GP1:90,2] + 37.873;
   1:L PR[91] R[100]mm/sec CNT100;
   1:  PR[GP1:91,1] = PR[GP1:90,1] + 28.507;
   1:  PR[GP1:91,2] = PR[GP1:90,2] + 37.914;
   1:L PR[91] R[100]mm/sec CNT100;
   1:  PR[GP1:91,1] = PR[GP1:90,1] + 21.891;
   1:  PR[GP1:91,2] = PR[GP1:90,2] + 37.946;
   1:L PR[91] R[100]mm/sec CNT100;
   1:  PR[GP1:91,1] = PR[GP1:90,1] + 14.841;
   1:  PR[GP1:91,2] = PR[GP1:90,2] + 38.074;
   1:L PR[91] R[100]mm/sec CNT100;
   1:  PR[GP1:91,1] = PR[GP1:90,1] + 14.242;
   1:  PR[GP1:91,2] = PR[GP1:90,2] + 38.053;
   1:L PR[91] R[100]mm/sec CNT100;
   1:  PR[GP1:91,1] = PR[GP1:90,1] + 12.309;
   1:  PR[GP1:91,2] = PR[GP1:90,2] + 37.455;
   1:L PR[91] R[100]mm/sec CNT100;
   1:  PR[GP1:91,1] = PR[GP1:90,1] + 7.406;
   1:  PR[GP1:91,2] = PR[GP1:90,2] + 35.872;
   1:L PR[91] R[100]mm/sec CNT100;
   1:  PR[GP1:91,1] = PR[GP1:90,1] + 2.543;
   1:  PR[GP1:91,2] = PR[GP1:90,2] + 34.292;
   1:L PR[91] R[100]mm/sec CNT100;
   1:  PR[GP1:91,1] = PR[GP1:90,1] + 2.270;
   1:  PR[GP1:91,2] = PR[GP1:90,2] + 34.140;
   1:L PR[91] R[100]mm/sec CNT100;
   1:  ! -- Layer/Ebene 120 -- !;
   1:  PR[91] = PR[90];
   1:  PR[GP1:91,1] = PR[GP1:90,1] + 1.930;
   1:  PR[GP1:91,2] = PR[GP1:90,2] + 34.414;
   1:  PR[GP1:91,3] = PR[GP1:90,3] + 73.505;
   1:L PR[91] R[100]mm/sec CNT100;
   1:  PR[GP1:91,1] = PR[GP1:90,1] + -2.078;
   1:  PR[GP1:91,2] = PR[GP1:90,2] + 34.389;
   1:L PR[91] R[100]mm/sec CNT100;
   1:  PR[GP1:91,1] = PR[GP1:90,1] + -10.832;
   1:  PR[GP1:91,2] = PR[GP1:90,2] + 37.245;
   1:L PR[91] R[100]mm/sec CNT100;
   1:  PR[GP1:91,1] = PR[GP1:90,1] + -13.735;
   1:  PR[GP1:91,2] = PR[GP1:90,2] + 38.142;
   1:L PR[91] R[100]mm/sec CNT100;
   1:  PR[GP1:91,1] = PR[GP1:90,1] + -14.669;
   1:  PR[GP1:91,2] = PR[GP1:90,2] + 38.176;
   1:L PR[91] R[100]mm/sec CNT100;
   1:  PR[GP1:91,1] = PR[GP1:90,1] + -25.132;
   1:  PR[GP1:91,2] = PR[GP1:90,2] + 37.985;
   1:L PR[91] R[100]mm/sec CNT100;
   1:  PR[GP1:91,1] = PR[GP1:90,1] + -28.111;
   1:  PR[GP1:91,2] = PR[GP1:90,2] + 37.970;
   1:L PR[91] R[100]mm/sec CNT100;
   1:  PR[GP1:91,1] = PR[GP1:90,1] + -28.144;
   1:  PR[GP1:91,2] = PR[GP1:90,2] + 37.963;
   1:L PR[91] R[100]mm/sec CNT100;
   1:  PR[GP1:91,1] = PR[GP1:90,1] + -41.272;
   1:  PR[GP1:91,2] = PR[GP1:90,2] + 33.295;
   1:L PR[91] R[100]mm/sec CNT100;
   1:  PR[GP1:91,1] = PR[GP1:90,1] + -41.811;
   1:  PR[GP1:91,2] = PR[GP1:90,2] + 32.960;
   1:L PR[91] R[100]mm/sec CNT100;
   1:  PR[GP1:91,1] = PR[GP1:90,1] + -42.392;
   1:  PR[GP1:91,2] = PR[GP1:90,2] + 32.443;
   1:L PR[91] R[100]mm/sec CNT100;
   1:  PR[GP1:91,1] = PR[GP1:90,1] + -52.004;
   1:  PR[GP1:91,2] = PR[GP1:90,2] + 24.665;
   1:L PR[91] R[100]mm/sec CNT100;
   1:  PR[GP1:91,1] = PR[GP1:90,1] + -52.685;
   1:  PR[GP1:91,2] = PR[GP1:90,2] + 23.778;
   1:L PR[91] R[100]mm/sec CNT100;
   1:  PR[GP1:91,1] = PR[GP1:90,1] + -53.295;
   1:  PR[GP1:91,2] = PR[GP1:90,2] + 22.595;
   1:L PR[91] R[100]mm/sec CNT100;
   1:  PR[GP1:91,1] = PR[GP1:90,1] + -59.035;
   1:  PR[GP1:91,2] = PR[GP1:90,2] + 13.007;
   1:L PR[91] R[100]mm/sec CNT100;
   1:  PR[GP1:91,1] = PR[GP1:90,1] + -59.431;
   1:  PR[GP1:91,2] = PR[GP1:90,2] + 11.665;
   1:L PR[91] R[100]mm/sec CNT100;
   1:  PR[GP1:91,1] = PR[GP1:90,1] + -59.568;
   1:  PR[GP1:91,2] = PR[GP1:90,2] + 10.161;
   1:L PR[91] R[100]mm/sec CNT100;
   1:  PR[GP1:91,1] = PR[GP1:90,1] + -61.460;
   1:  PR[GP1:91,2] = PR[GP1:90,2] + -0.100;
   1:L PR[91] R[100]mm/sec CNT100;
   1:  PR[GP1:91,1] = PR[GP1:90,1] + -61.320;
   1:  PR[GP1:91,2] = PR[GP1:90,2] + -1.641;
   1:L PR[91] R[100]mm/sec CNT100;
   1:  PR[GP1:91,1] = PR[GP1:90,1] + -59.437;
   1:  PR[GP1:91,2] = PR[GP1:90,2] + -11.785;
   1:L PR[91] R[100]mm/sec CNT100;
   1:  PR[GP1:91,1] = PR[GP1:90,1] + -59.028;
   1:  PR[GP1:91,2] = PR[GP1:90,2] + -13.173;
   1:L PR[91] R[100]mm/sec CNT100;
   1:  PR[GP1:91,1] = PR[GP1:90,1] + -58.363;
   1:  PR[GP1:91,2] = PR[GP1:90,2] + -14.478;
   1:L PR[91] R[100]mm/sec CNT100;
   1:  PR[GP1:91,1] = PR[GP1:90,1] + -52.692;
   1:  PR[GP1:91,2] = PR[GP1:90,2] + -23.913;
   1:L PR[91] R[100]mm/sec CNT100;
   1:  PR[GP1:91,1] = PR[GP1:90,1] + -51.990;
   1:  PR[GP1:91,2] = PR[GP1:90,2] + -24.827;
   1:L PR[91] R[100]mm/sec CNT100;
   1:  PR[GP1:91,1] = PR[GP1:90,1] + -51.194;
   1:  PR[GP1:91,2] = PR[GP1:90,2] + -25.541;
   1:L PR[91] R[100]mm/sec CNT100;
   1:  PR[GP1:91,1] = PR[GP1:90,1] + -41.812;
   1:  PR[GP1:91,2] = PR[GP1:90,2] + -33.102;
   1:L PR[91] R[100]mm/sec CNT100;
   1:  PR[GP1:91,1] = PR[GP1:90,1] + -41.251;
   1:  PR[GP1:91,2] = PR[GP1:90,2] + -33.452;
   1:L PR[91] R[100]mm/sec CNT100;
   1:  PR[GP1:91,1] = PR[GP1:90,1] + -40.692;
   1:  PR[GP1:91,2] = PR[GP1:90,2] + -33.676;
   1:L PR[91] R[100]mm/sec CNT100;
   1:  PR[GP1:91,1] = PR[GP1:90,1] + -28.126;
   1:  PR[GP1:91,2] = PR[GP1:90,2] + -38.110;
   1:L PR[91] R[100]mm/sec CNT100;
   1:  PR[GP1:91,1] = PR[GP1:90,1] + -28.084;
   1:  PR[GP1:91,2] = PR[GP1:90,2] + -38.119;
   1:L PR[91] R[100]mm/sec CNT100;
   1:  PR[GP1:91,1] = PR[GP1:90,1] + -28.028;
   1:  PR[GP1:91,2] = PR[GP1:90,2] + -38.121;
   1:L PR[91] R[100]mm/sec CNT100;
   1:  PR[GP1:91,1] = PR[GP1:90,1] + -25.133;
   1:  PR[GP1:91,2] = PR[GP1:90,2] + -38.130;
   1:L PR[91] R[100]mm/sec CNT100;
   1:  PR[GP1:91,1] = PR[GP1:90,1] + -14.650;
   1:  PR[GP1:91,2] = PR[GP1:90,2] + -38.316;
   1:L PR[91] R[100]mm/sec CNT100;
   1:  PR[GP1:91,1] = PR[GP1:90,1] + -13.715;
   1:  PR[GP1:91,2] = PR[GP1:90,2] + -38.283;
   1:L PR[91] R[100]mm/sec CNT100;
   1:  PR[GP1:91,1] = PR[GP1:90,1] + -10.174;
   1:  PR[GP1:91,2] = PR[GP1:90,2] + -37.180;
   1:L PR[91] R[100]mm/sec CNT100;
   1:  PR[GP1:91,1] = PR[GP1:90,1] + -2.079;
   1:  PR[GP1:91,2] = PR[GP1:90,2] + -34.539;
   1:L PR[91] R[100]mm/sec CNT100;
   1:  PR[GP1:91,1] = PR[GP1:90,1] + 2.273;
   1:  PR[GP1:91,2] = PR[GP1:90,2] + -34.549;
   1:L PR[91] R[100]mm/sec CNT100;
   1:  PR[GP1:91,1] = PR[GP1:90,1] + 10.381;
   1:  PR[GP1:91,2] = PR[GP1:90,2] + -37.178;
   1:L PR[91] R[100]mm/sec CNT100;
   1:  PR[GP1:91,1] = PR[GP1:90,1] + 13.925;
   1:  PR[GP1:91,2] = PR[GP1:90,2] + -38.282;
   1:L PR[91] R[100]mm/sec CNT100;
   1:  PR[GP1:91,1] = PR[GP1:90,1] + 14.860;
   1:  PR[GP1:91,2] = PR[GP1:90,2] + -38.316;
   1:L PR[91] R[100]mm/sec CNT100;
   1:  PR[GP1:91,1] = PR[GP1:90,1] + 25.345;
   1:  PR[GP1:91,2] = PR[GP1:90,2] + -38.131;
   1:L PR[91] R[100]mm/sec CNT100;
   1:  PR[GP1:91,1] = PR[GP1:90,1] + 28.304;
   1:  PR[GP1:91,2] = PR[GP1:90,2] + -38.118;
   1:L PR[91] R[100]mm/sec CNT100;
   1:  PR[GP1:91,1] = PR[GP1:90,1] + 28.335;
   1:  PR[GP1:91,2] = PR[GP1:90,2] + -38.111;
   1:L PR[91] R[100]mm/sec CNT100;
   1:  PR[GP1:91,1] = PR[GP1:90,1] + 41.470;
   1:  PR[GP1:91,2] = PR[GP1:90,2] + -33.450;
   1:L PR[91] R[100]mm/sec CNT100;
   1:  PR[GP1:91,1] = PR[GP1:90,1] + 42.005;
   1:  PR[GP1:91,2] = PR[GP1:90,2] + -33.119;
   1:L PR[91] R[100]mm/sec CNT100;
   1:  PR[GP1:91,1] = PR[GP1:90,1] + 42.582;
   1:  PR[GP1:91,2] = PR[GP1:90,2] + -32.607;
   1:L PR[91] R[100]mm/sec CNT100;
   1:  PR[GP1:91,1] = PR[GP1:90,1] + 52.197;
   1:  PR[GP1:91,2] = PR[GP1:90,2] + -24.825;
   1:L PR[91] R[100]mm/sec CNT100;
   1:  PR[GP1:91,1] = PR[GP1:90,1] + 52.886;
   1:  PR[GP1:91,2] = PR[GP1:90,2] + -23.930;
   1:L PR[91] R[100]mm/sec CNT100;
   1:  PR[GP1:91,1] = PR[GP1:90,1] + 53.498;
   1:  PR[GP1:91,2] = PR[GP1:90,2] + -22.757;
   1:L PR[91] R[100]mm/sec CNT100;
   1:  PR[GP1:91,1] = PR[GP1:90,1] + 59.241;
   1:  PR[GP1:91,2] = PR[GP1:90,2] + -13.187;
   1:L PR[91] R[100]mm/sec CNT100;
   1:  PR[GP1:91,1] = PR[GP1:90,1] + 59.636;
   1:  PR[GP1:91,2] = PR[GP1:90,2] + -11.866;
   1:L PR[91] R[100]mm/sec CNT100;
   1:  PR[GP1:91,1] = PR[GP1:90,1] + 59.780;
   1:  PR[GP1:91,2] = PR[GP1:90,2] + -10.321;
   1:L PR[91] R[100]mm/sec CNT100;
   1:  PR[GP1:91,1] = PR[GP1:90,1] + 61.673;
   1:  PR[GP1:91,2] = PR[GP1:90,2] + -0.045;
   1:L PR[91] R[100]mm/sec CNT100;
   1:  PR[GP1:91,1] = PR[GP1:90,1] + 61.526;
   1:  PR[GP1:91,2] = PR[GP1:90,2] + 1.542;
   1:L PR[91] R[100]mm/sec CNT100;
   1:  PR[GP1:91,1] = PR[GP1:90,1] + 59.645;
   1:  PR[GP1:91,2] = PR[GP1:90,2] + 11.693;
   1:L PR[91] R[100]mm/sec CNT100;
   1:  PR[GP1:91,1] = PR[GP1:90,1] + 59.237;
   1:  PR[GP1:91,2] = PR[GP1:90,2] + 13.059;
   1:L PR[91] R[100]mm/sec CNT100;
   1:  PR[GP1:91,1] = PR[GP1:90,1] + 58.569;
   1:  PR[GP1:91,2] = PR[GP1:90,2] + 14.352;
   1:L PR[91] R[100]mm/sec CNT100;
   1:  PR[GP1:91,1] = PR[GP1:90,1] + 52.902;
   1:  PR[GP1:91,2] = PR[GP1:90,2] + 23.766;
   1:L PR[91] R[100]mm/sec CNT100;
   1:  PR[GP1:91,1] = PR[GP1:90,1] + 52.192;
   1:  PR[GP1:91,2] = PR[GP1:90,2] + 24.687;
   1:L PR[91] R[100]mm/sec CNT100;
   1:  PR[GP1:91,1] = PR[GP1:90,1] + 51.401;
   1:  PR[GP1:91,2] = PR[GP1:90,2] + 25.395;
   1:L PR[91] R[100]mm/sec CNT100;
   1:  PR[GP1:91,1] = PR[GP1:90,1] + 42.027;
   1:  PR[GP1:91,2] = PR[GP1:90,2] + 32.962;
   1:L PR[91] R[100]mm/sec CNT100;
   1:  PR[GP1:91,1] = PR[GP1:90,1] + 41.471;
   1:  PR[GP1:91,2] = PR[GP1:90,2] + 33.307;
   1:L PR[91] R[100]mm/sec CNT100;
   1:  PR[GP1:91,1] = PR[GP1:90,1] + 40.910;
   1:  PR[GP1:91,2] = PR[GP1:90,2] + 33.531;
   1:L PR[91] R[100]mm/sec CNT100;
   1:  PR[GP1:91,1] = PR[GP1:90,1] + 28.353;
   1:  PR[GP1:91,2] = PR[GP1:90,2] + 37.964;
   1:L PR[91] R[100]mm/sec CNT100;
   1:  PR[GP1:91,1] = PR[GP1:90,1] + 28.320;
   1:  PR[GP1:91,2] = PR[GP1:90,2] + 37.971;
   1:L PR[91] R[100]mm/sec CNT100;
   1:  PR[GP1:91,1] = PR[GP1:90,1] + 25.345;
   1:  PR[GP1:91,2] = PR[GP1:90,2] + 37.985;
   1:L PR[91] R[100]mm/sec CNT100;
   1:  PR[GP1:91,1] = PR[GP1:90,1] + 14.879;
   1:  PR[GP1:91,2] = PR[GP1:90,2] + 38.175;
   1:L PR[91] R[100]mm/sec CNT100;
   1:  PR[GP1:91,1] = PR[GP1:90,1] + 13.945;
   1:  PR[GP1:91,2] = PR[GP1:90,2] + 38.141;
   1:L PR[91] R[100]mm/sec CNT100;
   1:  PR[GP1:91,1] = PR[GP1:90,1] + 11.039;
   1:  PR[GP1:91,2] = PR[GP1:90,2] + 37.243;
   1:L PR[91] R[100]mm/sec CNT100;
   1:  PR[GP1:91,1] = PR[GP1:90,1] + 3.764;
   1:  PR[GP1:91,2] = PR[GP1:90,2] + 34.895;
   1:L PR[91] R[100]mm/sec CNT100;
   1:  PR[GP1:91,1] = PR[GP1:90,1] + 2.241;
   1:  PR[GP1:91,2] = PR[GP1:90,2] + 34.388;
   1:L PR[91] R[100]mm/sec CNT100;
   1:  ! -- Layer/Ebene 121 -- !;
   1:  PR[91] = PR[90];
   1:  PR[GP1:91,1] = PR[GP1:90,1] + -2.051;
   1:  PR[GP1:91,2] = PR[GP1:90,2] + 34.583;
   1:  PR[GP1:91,3] = PR[GP1:90,3] + 74.115;
   1:L PR[91] R[100]mm/sec CNT100;
   1:  PR[GP1:91,1] = PR[GP1:90,1] + -9.562;
   1:  PR[GP1:91,2] = PR[GP1:90,2] + 37.033;
   1:L PR[91] R[100]mm/sec CNT100;
   1:  PR[GP1:91,1] = PR[GP1:90,1] + -13.438;
   1:  PR[GP1:91,2] = PR[GP1:90,2] + 38.231;
   1:L PR[91] R[100]mm/sec CNT100;
   1:  PR[GP1:91,1] = PR[GP1:90,1] + -14.708;
   1:  PR[GP1:91,2] = PR[GP1:90,2] + 38.276;
   1:L PR[91] R[100]mm/sec CNT100;
   1:  PR[GP1:91,1] = PR[GP1:90,1] + -27.868;
   1:  PR[GP1:91,2] = PR[GP1:90,2] + 38.036;
   1:L PR[91] R[100]mm/sec CNT100;
   1:  PR[GP1:91,1] = PR[GP1:90,1] + -41.089;
   1:  PR[GP1:91,2] = PR[GP1:90,2] + 33.335;
   1:L PR[91] R[100]mm/sec CNT100;
   1:  PR[GP1:91,1] = PR[GP1:90,1] + -41.486;
   1:  PR[GP1:91,2] = PR[GP1:90,2] + 33.088;
   1:L PR[91] R[100]mm/sec CNT100;
   1:  PR[GP1:91,1] = PR[GP1:90,1] + -41.932;
   1:  PR[GP1:91,2] = PR[GP1:90,2] + 32.692;
   1:L PR[91] R[100]mm/sec CNT100;
   1:  PR[GP1:91,1] = PR[GP1:90,1] + -51.820;
   1:  PR[GP1:91,2] = PR[GP1:90,2] + 24.690;
   1:L PR[91] R[100]mm/sec CNT100;
   1:  PR[GP1:91,1] = PR[GP1:90,1] + -52.401;
   1:  PR[GP1:91,2] = PR[GP1:90,2] + 23.934;
   1:L PR[91] R[100]mm/sec CNT100;
   1:  PR[GP1:91,1] = PR[GP1:90,1] + -52.927;
   1:  PR[GP1:91,2] = PR[GP1:90,2] + 22.913;
   1:L PR[91] R[100]mm/sec CNT100;
   1:  PR[GP1:91,1] = PR[GP1:90,1] + -58.848;
   1:  PR[GP1:91,2] = PR[GP1:90,2] + 13.022;
   1:L PR[91] R[100]mm/sec CNT100;
   1:  PR[GP1:91,1] = PR[GP1:90,1] + -59.198;
   1:  PR[GP1:91,2] = PR[GP1:90,2] + 11.836;
   1:L PR[91] R[100]mm/sec CNT100;
   1:  PR[GP1:91,1] = PR[GP1:90,1] + -59.320;
   1:  PR[GP1:91,2] = PR[GP1:90,2] + 10.495;
   1:L PR[91] R[100]mm/sec CNT100;
   1:  PR[GP1:91,1] = PR[GP1:90,1] + -61.273;
   1:  PR[GP1:91,2] = PR[GP1:90,2] + -0.100;
   1:L PR[91] R[100]mm/sec CNT100;
   1:  PR[GP1:91,1] = PR[GP1:90,1] + -61.148;
   1:  PR[GP1:91,2] = PR[GP1:90,2] + -1.485;
   1:L PR[91] R[100]mm/sec CNT100;
   1:  PR[GP1:91,1] = PR[GP1:90,1] + -59.204;
   1:  PR[GP1:91,2] = PR[GP1:90,2] + -11.957;
   1:L PR[91] R[100]mm/sec CNT100;
   1:  PR[GP1:91,1] = PR[GP1:90,1] + -58.841;
   1:  PR[GP1:91,2] = PR[GP1:90,2] + -13.189;
   1:L PR[91] R[100]mm/sec CNT100;
   1:  PR[GP1:91,1] = PR[GP1:90,1] + -58.250;
   1:  PR[GP1:91,2] = PR[GP1:90,2] + -14.348;
   1:L PR[91] R[100]mm/sec CNT100;
   1:  PR[GP1:91,1] = PR[GP1:90,1] + -52.407;
   1:  PR[GP1:91,2] = PR[GP1:90,2] + -24.069;
   1:L PR[91] R[100]mm/sec CNT100;
   1:  PR[GP1:91,1] = PR[GP1:90,1] + -51.806;
   1:  PR[GP1:91,2] = PR[GP1:90,2] + -24.851;
   1:L PR[91] R[100]mm/sec CNT100;
   1:  PR[GP1:91,1] = PR[GP1:90,1] + -51.124;
   1:  PR[GP1:91,2] = PR[GP1:90,2] + -25.463;
   1:L PR[91] R[100]mm/sec CNT100;
   1:  PR[GP1:91,1] = PR[GP1:90,1] + -41.487;
   1:  PR[GP1:91,2] = PR[GP1:90,2] + -33.231;
   1:L PR[91] R[100]mm/sec CNT100;
   1:  PR[GP1:91,1] = PR[GP1:90,1] + -41.067;
   1:  PR[GP1:91,2] = PR[GP1:90,2] + -33.492;
   1:L PR[91] R[100]mm/sec CNT100;
   1:  PR[GP1:91,1] = PR[GP1:90,1] + -40.646;
   1:  PR[GP1:91,2] = PR[GP1:90,2] + -33.661;
   1:L PR[91] R[100]mm/sec CNT100;
   1:  PR[GP1:91,1] = PR[GP1:90,1] + -27.850;
   1:  PR[GP1:91,2] = PR[GP1:90,2] + -38.184;
   1:L PR[91] R[100]mm/sec CNT100;
   1:  PR[GP1:91,1] = PR[GP1:90,1] + -14.690;
   1:  PR[GP1:91,2] = PR[GP1:90,2] + -38.417;
   1:L PR[91] R[100]mm/sec CNT100;
   1:  PR[GP1:91,1] = PR[GP1:90,1] + -13.392;
   1:  PR[GP1:91,2] = PR[GP1:90,2] + -38.365;
   1:L PR[91] R[100]mm/sec CNT100;
   1:  PR[GP1:91,1] = PR[GP1:90,1] + -8.698;
   1:  PR[GP1:91,2] = PR[GP1:90,2] + -36.902;
   1:L PR[91] R[100]mm/sec CNT100;
   1:  PR[GP1:91,1] = PR[GP1:90,1] + -2.052;
   1:  PR[GP1:91,2] = PR[GP1:90,2] + -34.733;
   1:L PR[91] R[100]mm/sec CNT100;
   1:  PR[GP1:91,1] = PR[GP1:90,1] + 0.528;
   1:L PR[91] R[100]mm/sec CNT100;
   1:  PR[GP1:91,1] = PR[GP1:90,1] + 2.261;
   1:  PR[GP1:91,2] = PR[GP1:90,2] + -34.751;
   1:L PR[91] R[100]mm/sec CNT100;
   1:  PR[GP1:91,1] = PR[GP1:90,1] + 8.905;
   1:  PR[GP1:91,2] = PR[GP1:90,2] + -36.900;
   1:L PR[91] R[100]mm/sec CNT100;
   1:  PR[GP1:91,1] = PR[GP1:90,1] + 13.628;
   1:  PR[GP1:91,2] = PR[GP1:90,2] + -38.371;
   1:L PR[91] R[100]mm/sec CNT100;
   1:  PR[GP1:91,1] = PR[GP1:90,1] + 14.899;
   1:  PR[GP1:91,2] = PR[GP1:90,2] + -38.416;
   1:L PR[91] R[100]mm/sec CNT100;
   1:  PR[GP1:91,1] = PR[GP1:90,1] + 28.060;
   1:  PR[GP1:91,2] = PR[GP1:90,2] + -38.184;
   1:L PR[91] R[100]mm/sec CNT100;
   1:  PR[GP1:91,1] = PR[GP1:90,1] + 41.288;
   1:  PR[GP1:91,2] = PR[GP1:90,2] + -33.490;
   1:L PR[91] R[100]mm/sec CNT100;
   1:  PR[GP1:91,1] = PR[GP1:90,1] + 41.681;
   1:  PR[GP1:91,2] = PR[GP1:90,2] + -33.246;
   1:L PR[91] R[100]mm/sec CNT100;
   1:  PR[GP1:91,1] = PR[GP1:90,1] + 42.124;
   1:  PR[GP1:91,2] = PR[GP1:90,2] + -32.854;
   1:L PR[91] R[100]mm/sec CNT100;
   1:  PR[GP1:91,1] = PR[GP1:90,1] + 52.015;
   1:  PR[GP1:91,2] = PR[GP1:90,2] + -24.847;
   1:L PR[91] R[100]mm/sec CNT100;
   1:  PR[GP1:91,1] = PR[GP1:90,1] + 52.603;
   1:  PR[GP1:91,2] = PR[GP1:90,2] + -24.085;
   1:L PR[91] R[100]mm/sec CNT100;
   1:  PR[GP1:91,1] = PR[GP1:90,1] + 53.130;
   1:  PR[GP1:91,2] = PR[GP1:90,2] + -23.072;
   1:L PR[91] R[100]mm/sec CNT100;
   1:  PR[GP1:91,1] = PR[GP1:90,1] + 59.055;
   1:  PR[GP1:91,2] = PR[GP1:90,2] + -13.201;
   1:L PR[91] R[100]mm/sec CNT100;
   1:  PR[GP1:91,1] = PR[GP1:90,1] + 59.404;
   1:  PR[GP1:91,2] = PR[GP1:90,2] + -12.034;
   1:L PR[91] R[100]mm/sec CNT100;
   1:  PR[GP1:91,1] = PR[GP1:90,1] + 59.532;
   1:  PR[GP1:91,2] = PR[GP1:90,2] + -10.656;
   1:L PR[91] R[100]mm/sec CNT100;
   1:  PR[GP1:91,1] = PR[GP1:90,1] + 61.486;
   1:  PR[GP1:91,2] = PR[GP1:90,2] + -0.045;
   1:L PR[91] R[100]mm/sec CNT100;
   1:  PR[GP1:91,1] = PR[GP1:90,1] + 61.355;
   1:  PR[GP1:91,2] = PR[GP1:90,2] + 1.381;
   1:L PR[91] R[100]mm/sec CNT100;
   1:  PR[GP1:91,1] = PR[GP1:90,1] + 59.413;
   1:  PR[GP1:91,2] = PR[GP1:90,2] + 11.861;
   1:L PR[91] R[100]mm/sec CNT100;
   1:  PR[GP1:91,1] = PR[GP1:90,1] + 59.051;
   1:  PR[GP1:91,2] = PR[GP1:90,2] + 13.073;
   1:L PR[91] R[100]mm/sec CNT100;
   1:  PR[GP1:91,1] = PR[GP1:90,1] + 58.457;
   1:  PR[GP1:91,2] = PR[GP1:90,2] + 14.222;
   1:L PR[91] R[100]mm/sec CNT100;
   1:  PR[GP1:91,1] = PR[GP1:90,1] + 52.619;
   1:  PR[GP1:91,2] = PR[GP1:90,2] + 23.920;
   1:L PR[91] R[100]mm/sec CNT100;
   1:  PR[GP1:91,1] = PR[GP1:90,1] + 52.011;
   1:  PR[GP1:91,2] = PR[GP1:90,2] + 24.709;
   1:L PR[91] R[100]mm/sec CNT100;
   1:  PR[GP1:91,1] = PR[GP1:90,1] + 51.332;
   1:  PR[GP1:91,2] = PR[GP1:90,2] + 25.316;
   1:L PR[91] R[100]mm/sec CNT100;
   1:  PR[GP1:91,1] = PR[GP1:90,1] + 41.704;
   1:  PR[GP1:91,2] = PR[GP1:90,2] + 33.089;
   1:L PR[91] R[100]mm/sec CNT100;
   1:  PR[GP1:91,1] = PR[GP1:90,1] + 41.288;
   1:  PR[GP1:91,2] = PR[GP1:90,2] + 33.346;
   1:L PR[91] R[100]mm/sec CNT100;
   1:  PR[GP1:91,1] = PR[GP1:90,1] + 40.865;
   1:  PR[GP1:91,2] = PR[GP1:90,2] + 33.515;
   1:L PR[91] R[100]mm/sec CNT100;
   1:  PR[GP1:91,1] = PR[GP1:90,1] + 28.078;
   1:  PR[GP1:91,2] = PR[GP1:90,2] + 38.037;
   1:L PR[91] R[100]mm/sec CNT100;
   1:  PR[GP1:91,1] = PR[GP1:90,1] + 14.918;
   1:  PR[GP1:91,2] = PR[GP1:90,2] + 38.275;
   1:L PR[91] R[100]mm/sec CNT100;
   1:  PR[GP1:91,1] = PR[GP1:90,1] + 13.647;
   1:  PR[GP1:91,2] = PR[GP1:90,2] + 38.230;
   1:L PR[91] R[100]mm/sec CNT100;
   1:  PR[GP1:91,1] = PR[GP1:90,1] + 9.769;
   1:  PR[GP1:91,2] = PR[GP1:90,2] + 37.031;
   1:L PR[91] R[100]mm/sec CNT100;
   1:  PR[GP1:91,1] = PR[GP1:90,1] + 2.259;
   1:  PR[GP1:91,2] = PR[GP1:90,2] + 34.607;
   1:L PR[91] R[100]mm/sec CNT100;
   1:  ! -- Layer/Ebene 122 -- !;
   1:  PR[91] = PR[90];
   1:  PR[GP1:91,1] = PR[GP1:90,1] + -2.024;
   1:  PR[GP1:91,2] = PR[GP1:90,2] + 34.777;
   1:  PR[GP1:91,3] = PR[GP1:90,3] + 74.725;
   1:L PR[91] R[100]mm/sec CNT100;
   1:  PR[GP1:91,1] = PR[GP1:90,1] + -8.291;
   1:  PR[GP1:91,2] = PR[GP1:90,2] + 36.821;
   1:L PR[91] R[100]mm/sec CNT100;
   1:  PR[GP1:91,1] = PR[GP1:90,1] + -13.140;
   1:  PR[GP1:91,2] = PR[GP1:90,2] + 38.320;
   1:L PR[91] R[100]mm/sec CNT100;
   1:  PR[GP1:91,1] = PR[GP1:90,1] + -14.746;
   1:  PR[GP1:91,2] = PR[GP1:90,2] + 38.377;
   1:L PR[91] R[100]mm/sec CNT100;
   1:  PR[GP1:91,1] = PR[GP1:90,1] + -27.614;
   1:  PR[GP1:91,2] = PR[GP1:90,2] + 38.142;
   1:L PR[91] R[100]mm/sec CNT100;
   1:  PR[GP1:91,1] = PR[GP1:90,1] + -27.902;
   1:  PR[GP1:91,2] = PR[GP1:90,2] + 38.048;
   1:L PR[91] R[100]mm/sec CNT100;
   1:  PR[GP1:91,1] = PR[GP1:90,1] + -31.851;
   1:  PR[GP1:91,2] = PR[GP1:90,2] + 36.590;
   1:L PR[91] R[100]mm/sec CNT100;
   1:  PR[GP1:91,1] = PR[GP1:90,1] + -40.905;
   1:  PR[GP1:91,2] = PR[GP1:90,2] + 33.375;
   1:L PR[91] R[100]mm/sec CNT100;
   1:  PR[GP1:91,1] = PR[GP1:90,1] + -41.161;
   1:  PR[GP1:91,2] = PR[GP1:90,2] + 33.216;
   1:L PR[91] R[100]mm/sec CNT100;
   1:  PR[GP1:91,1] = PR[GP1:90,1] + -41.472;
   1:  PR[GP1:91,2] = PR[GP1:90,2] + 32.940;
   1:L PR[91] R[100]mm/sec CNT100;
   1:  PR[GP1:91,1] = PR[GP1:90,1] + -51.637;
   1:  PR[GP1:91,2] = PR[GP1:90,2] + 24.714;
   1:L PR[91] R[100]mm/sec CNT100;
   1:  PR[GP1:91,1] = PR[GP1:90,1] + -52.116;
   1:  PR[GP1:91,2] = PR[GP1:90,2] + 24.090;
   1:L PR[91] R[100]mm/sec CNT100;
   1:  PR[GP1:91,1] = PR[GP1:90,1] + -52.559;
   1:  PR[GP1:91,2] = PR[GP1:90,2] + 23.232;
   1:L PR[91] R[100]mm/sec CNT100;
   1:  PR[GP1:91,1] = PR[GP1:90,1] + -58.661;
   1:  PR[GP1:91,2] = PR[GP1:90,2] + 13.038;
   1:L PR[91] R[100]mm/sec CNT100;
   1:  PR[GP1:91,1] = PR[GP1:90,1] + -58.965;
   1:  PR[GP1:91,2] = PR[GP1:90,2] + 12.008;
   1:L PR[91] R[100]mm/sec CNT100;
   1:  PR[GP1:91,1] = PR[GP1:90,1] + -59.072;
   1:  PR[GP1:91,2] = PR[GP1:90,2] + 10.830;
   1:L PR[91] R[100]mm/sec CNT100;
   1:  PR[GP1:91,1] = PR[GP1:90,1] + -61.087;
   1:  PR[GP1:91,2] = PR[GP1:90,2] + -0.100;
   1:L PR[91] R[100]mm/sec CNT100;
   1:  PR[GP1:91,1] = PR[GP1:90,1] + -60.976;
   1:  PR[GP1:91,2] = PR[GP1:90,2] + -1.328;
   1:L PR[91] R[100]mm/sec CNT100;
   1:  PR[GP1:91,1] = PR[GP1:90,1] + -58.971;
   1:  PR[GP1:91,2] = PR[GP1:90,2] + -12.129;
   1:L PR[91] R[100]mm/sec CNT100;
   1:  PR[GP1:91,1] = PR[GP1:90,1] + -58.654;
   1:  PR[GP1:91,2] = PR[GP1:90,2] + -13.205;
   1:L PR[91] R[100]mm/sec CNT100;
   1:  PR[GP1:91,1] = PR[GP1:90,1] + -58.137;
   1:  PR[GP1:91,2] = PR[GP1:90,2] + -14.218;
   1:L PR[91] R[100]mm/sec CNT100;
   1:  PR[GP1:91,1] = PR[GP1:90,1] + -52.123;
   1:  PR[GP1:91,2] = PR[GP1:90,2] + -24.225;
   1:L PR[91] R[100]mm/sec CNT100;
   1:  PR[GP1:91,1] = PR[GP1:90,1] + -51.623;
   1:  PR[GP1:91,2] = PR[GP1:90,2] + -24.876;
   1:L PR[91] R[100]mm/sec CNT100;
   1:  PR[GP1:91,1] = PR[GP1:90,1] + -51.054;
   1:  PR[GP1:91,2] = PR[GP1:90,2] + -25.386;
   1:L PR[91] R[100]mm/sec CNT100;
   1:  PR[GP1:91,1] = PR[GP1:90,1] + -41.161;
   1:  PR[GP1:91,2] = PR[GP1:90,2] + -33.359;
   1:L PR[91] R[100]mm/sec CNT100;
   1:  PR[GP1:91,1] = PR[GP1:90,1] + -40.884;
   1:  PR[GP1:91,2] = PR[GP1:90,2] + -33.532;
   1:L PR[91] R[100]mm/sec CNT100;
   1:  PR[GP1:91,1] = PR[GP1:90,1] + -40.600;
   1:  PR[GP1:91,2] = PR[GP1:90,2] + -33.646;
   1:L PR[91] R[100]mm/sec CNT100;
   1:  PR[GP1:91,1] = PR[GP1:90,1] + -31.852;
   1:  PR[GP1:91,2] = PR[GP1:90,2] + -36.733;
   1:L PR[91] R[100]mm/sec CNT100;
   1:  PR[GP1:91,1] = PR[GP1:90,1] + -27.886;
   1:  PR[GP1:91,2] = PR[GP1:90,2] + -38.194;
   1:L PR[91] R[100]mm/sec CNT100;
   1:  PR[GP1:91,1] = PR[GP1:90,1] + -27.596;
   1:  PR[GP1:91,2] = PR[GP1:90,2] + -38.289;
   1:L PR[91] R[100]mm/sec CNT100;
   1:  PR[GP1:91,1] = PR[GP1:90,1] + -14.729;
   1:  PR[GP1:91,2] = PR[GP1:90,2] + -38.518;
   1:L PR[91] R[100]mm/sec CNT100;
   1:  PR[GP1:91,1] = PR[GP1:90,1] + -13.088;
   1:  PR[GP1:91,2] = PR[GP1:90,2] + -38.452;
   1:L PR[91] R[100]mm/sec CNT100;
   1:  PR[GP1:91,1] = PR[GP1:90,1] + -7.223;
   1:  PR[GP1:91,2] = PR[GP1:90,2] + -36.624;
   1:L PR[91] R[100]mm/sec CNT100;
   1:  PR[GP1:91,1] = PR[GP1:90,1] + -2.024;
   1:  PR[GP1:91,2] = PR[GP1:90,2] + -34.928;
   1:L PR[91] R[100]mm/sec CNT100;
   1:  PR[GP1:91,1] = PR[GP1:90,1] + 2.232;
   1:  PR[GP1:91,2] = PR[GP1:90,2] + -34.941;
   1:L PR[91] R[100]mm/sec CNT100;
   1:  PR[GP1:91,1] = PR[GP1:90,1] + 7.429;
   1:  PR[GP1:91,2] = PR[GP1:90,2] + -36.622;
   1:L PR[91] R[100]mm/sec CNT100;
   1:  PR[GP1:91,1] = PR[GP1:90,1] + 13.332;
   1:  PR[GP1:91,2] = PR[GP1:90,2] + -38.460;
   1:L PR[91] R[100]mm/sec CNT100;
   1:  PR[GP1:91,1] = PR[GP1:90,1] + 14.938;
   1:  PR[GP1:91,2] = PR[GP1:90,2] + -38.517;
   1:L PR[91] R[100]mm/sec CNT100;
   1:  PR[GP1:91,1] = PR[GP1:90,1] + 27.807;
   1:  PR[GP1:91,2] = PR[GP1:90,2] + -38.290;
   1:L PR[91] R[100]mm/sec CNT100;
   1:  PR[GP1:91,1] = PR[GP1:90,1] + 28.097;
   1:  PR[GP1:91,2] = PR[GP1:90,2] + -38.195;
   1:L PR[91] R[100]mm/sec CNT100;
   1:  PR[GP1:91,1] = PR[GP1:90,1] + 32.063;
   1:  PR[GP1:91,2] = PR[GP1:90,2] + -36.734;
   1:L PR[91] R[100]mm/sec CNT100;
   1:  PR[GP1:91,1] = PR[GP1:90,1] + 41.105;
   1:  PR[GP1:91,2] = PR[GP1:90,2] + -33.530;
   1:L PR[91] R[100]mm/sec CNT100;
   1:  PR[GP1:91,1] = PR[GP1:90,1] + 41.358;
   1:  PR[GP1:91,2] = PR[GP1:90,2] + -33.373;
   1:L PR[91] R[100]mm/sec CNT100;
   1:  PR[GP1:91,1] = PR[GP1:90,1] + 41.666;
   1:  PR[GP1:91,2] = PR[GP1:90,2] + -33.100;
   1:L PR[91] R[100]mm/sec CNT100;
   1:  PR[GP1:91,1] = PR[GP1:90,1] + 51.834;
   1:  PR[GP1:91,2] = PR[GP1:90,2] + -24.869;
   1:L PR[91] R[100]mm/sec CNT100;
   1:  PR[GP1:91,1] = PR[GP1:90,1] + 52.319;
   1:  PR[GP1:91,2] = PR[GP1:90,2] + -24.240;
   1:L PR[91] R[100]mm/sec CNT100;
   1:  PR[GP1:91,1] = PR[GP1:90,1] + 52.762;
   1:  PR[GP1:91,2] = PR[GP1:90,2] + -23.388;
   1:L PR[91] R[100]mm/sec CNT100;
   1:  PR[GP1:91,1] = PR[GP1:90,1] + 58.868;
   1:  PR[GP1:91,2] = PR[GP1:90,2] + -13.215;
   1:L PR[91] R[100]mm/sec CNT100;
   1:  PR[GP1:91,1] = PR[GP1:90,1] + 59.171;
   1:  PR[GP1:91,2] = PR[GP1:90,2] + -12.202;
   1:L PR[91] R[100]mm/sec CNT100;
   1:  PR[GP1:91,1] = PR[GP1:90,1] + 59.284;
   1:  PR[GP1:91,2] = PR[GP1:90,2] + -10.991;
   1:L PR[91] R[100]mm/sec CNT100;
   1:  PR[GP1:91,1] = PR[GP1:90,1] + 61.300;
   1:  PR[GP1:91,2] = PR[GP1:90,2] + -0.045;
   1:L PR[91] R[100]mm/sec CNT100;
   1:  PR[GP1:91,1] = PR[GP1:90,1] + 61.183;
   1:  PR[GP1:91,2] = PR[GP1:90,2] + 1.220;
   1:L PR[91] R[100]mm/sec CNT100;
   1:  PR[GP1:91,1] = PR[GP1:90,1] + 59.180;
   1:  PR[GP1:91,2] = PR[GP1:90,2] + 12.028;
   1:L PR[91] R[100]mm/sec CNT100;
   1:  PR[GP1:91,1] = PR[GP1:90,1] + 58.864;
   1:  PR[GP1:91,2] = PR[GP1:90,2] + 13.087;
   1:L PR[91] R[100]mm/sec CNT100;
   1:  PR[GP1:91,1] = PR[GP1:90,1] + 58.346;
   1:  PR[GP1:91,2] = PR[GP1:90,2] + 14.092;
   1:L PR[91] R[100]mm/sec CNT100;
   1:  PR[GP1:91,1] = PR[GP1:90,1] + 52.335;
   1:  PR[GP1:91,2] = PR[GP1:90,2] + 24.075;
   1:L PR[91] R[100]mm/sec CNT100;
   1:  PR[GP1:91,1] = PR[GP1:90,1] + 51.830;
   1:  PR[GP1:91,2] = PR[GP1:90,2] + 24.731;
   1:L PR[91] R[100]mm/sec CNT100;
   1:  PR[GP1:91,1] = PR[GP1:90,1] + 51.264;
   1:  PR[GP1:91,2] = PR[GP1:90,2] + 25.238;
   1:L PR[91] R[100]mm/sec CNT100;
   1:  PR[GP1:91,1] = PR[GP1:90,1] + 41.380;
   1:  PR[GP1:91,2] = PR[GP1:90,2] + 33.215;
   1:L PR[91] R[100]mm/sec CNT100;
   1:  PR[GP1:91,1] = PR[GP1:90,1] + 41.105;
   1:  PR[GP1:91,2] = PR[GP1:90,2] + 33.386;
   1:L PR[91] R[100]mm/sec CNT100;
   1:  PR[GP1:91,1] = PR[GP1:90,1] + 40.821;
   1:  PR[GP1:91,2] = PR[GP1:90,2] + 33.500;
   1:L PR[91] R[100]mm/sec CNT100;
   1:  PR[GP1:91,1] = PR[GP1:90,1] + 32.064;
   1:  PR[GP1:91,2] = PR[GP1:90,2] + 36.591;
   1:L PR[91] R[100]mm/sec CNT100;
   1:  PR[GP1:91,1] = PR[GP1:90,1] + 28.113;
   1:  PR[GP1:91,2] = PR[GP1:90,2] + 38.048;
   1:L PR[91] R[100]mm/sec CNT100;
   1:  PR[GP1:91,1] = PR[GP1:90,1] + 27.824;
   1:  PR[GP1:91,2] = PR[GP1:90,2] + 38.143;
   1:L PR[91] R[100]mm/sec CNT100;
   1:  PR[GP1:91,1] = PR[GP1:90,1] + 14.956;
   1:  PR[GP1:91,2] = PR[GP1:90,2] + 38.376;
   1:L PR[91] R[100]mm/sec CNT100;
   1:  PR[GP1:91,1] = PR[GP1:90,1] + 13.350;
   1:  PR[GP1:91,2] = PR[GP1:90,2] + 38.319;
   1:L PR[91] R[100]mm/sec CNT100;
   1:  PR[GP1:91,1] = PR[GP1:90,1] + 8.499;
   1:  PR[GP1:91,2] = PR[GP1:90,2] + 36.819;
   1:L PR[91] R[100]mm/sec CNT100;
   1:  PR[GP1:91,1] = PR[GP1:90,1] + 2.233;
   1:  PR[GP1:91,2] = PR[GP1:90,2] + 34.796;
   1:L PR[91] R[100]mm/sec CNT100;
   1:  ! -- Layer/Ebene 123 -- !;
   1:  PR[91] = PR[90];
   1:  PR[GP1:91,1] = PR[GP1:90,1] + -1.997;
   1:  PR[GP1:91,2] = PR[GP1:90,2] + 34.970;
   1:  PR[GP1:91,3] = PR[GP1:90,3] + 75.335;
   1:L PR[91] R[100]mm/sec CNT100;
   1:  PR[GP1:91,1] = PR[GP1:90,1] + -7.021;
   1:  PR[GP1:91,2] = PR[GP1:90,2] + 36.609;
   1:L PR[91] R[100]mm/sec CNT100;
   1:  PR[GP1:91,1] = PR[GP1:90,1] + -12.843;
   1:  PR[GP1:91,2] = PR[GP1:90,2] + 38.408;
   1:L PR[91] R[100]mm/sec CNT100;
   1:  PR[GP1:91,1] = PR[GP1:90,1] + -14.784;
   1:  PR[GP1:91,2] = PR[GP1:90,2] + 38.478;
   1:L PR[91] R[100]mm/sec CNT100;
   1:  PR[GP1:91,1] = PR[GP1:90,1] + -27.353;
   1:  PR[GP1:91,2] = PR[GP1:90,2] + 38.248;
   1:L PR[91] R[100]mm/sec CNT100;
   1:  PR[GP1:91,1] = PR[GP1:90,1] + -27.971;
   1:  PR[GP1:91,2] = PR[GP1:90,2] + 38.046;
   1:L PR[91] R[100]mm/sec CNT100;
   1:  PR[GP1:91,1] = PR[GP1:90,1] + -35.312;
   1:  PR[GP1:91,2] = PR[GP1:90,2] + 35.336;
   1:L PR[91] R[100]mm/sec CNT100;
   1:  PR[GP1:91,1] = PR[GP1:90,1] + -40.722;
   1:  PR[GP1:91,2] = PR[GP1:90,2] + 33.415;
   1:L PR[91] R[100]mm/sec CNT100;
   1:  PR[GP1:91,1] = PR[GP1:90,1] + -40.836;
   1:  PR[GP1:91,2] = PR[GP1:90,2] + 33.344;
   1:L PR[91] R[100]mm/sec CNT100;
   1:  PR[GP1:91,1] = PR[GP1:90,1] + -41.011;
   1:  PR[GP1:91,2] = PR[GP1:90,2] + 33.189;
   1:L PR[91] R[100]mm/sec CNT100;
   1:  PR[GP1:91,1] = PR[GP1:90,1] + -51.454;
   1:  PR[GP1:91,2] = PR[GP1:90,2] + 24.738;
   1:L PR[91] R[100]mm/sec CNT100;
   1:  PR[GP1:91,1] = PR[GP1:90,1] + -51.831;
   1:  PR[GP1:91,2] = PR[GP1:90,2] + 24.246;
   1:L PR[91] R[100]mm/sec CNT100;
   1:  PR[GP1:91,1] = PR[GP1:90,1] + -52.190;
   1:  PR[GP1:91,2] = PR[GP1:90,2] + 23.550;
   1:L PR[91] R[100]mm/sec CNT100;
   1:  PR[GP1:91,1] = PR[GP1:90,1] + -58.474;
   1:  PR[GP1:91,2] = PR[GP1:90,2] + 13.053;
   1:L PR[91] R[100]mm/sec CNT100;
   1:  PR[GP1:91,1] = PR[GP1:90,1] + -58.732;
   1:  PR[GP1:91,2] = PR[GP1:90,2] + 12.180;
   1:L PR[91] R[100]mm/sec CNT100;
   1:  PR[GP1:91,1] = PR[GP1:90,1] + -58.825;
   1:  PR[GP1:91,2] = PR[GP1:90,2] + 11.164;
   1:L PR[91] R[100]mm/sec CNT100;
   1:  PR[GP1:91,1] = PR[GP1:90,1] + -60.901;
   1:  PR[GP1:91,2] = PR[GP1:90,2] + -0.100;
   1:L PR[91] R[100]mm/sec CNT100;
   1:  PR[GP1:91,1] = PR[GP1:90,1] + -60.804;
   1:  PR[GP1:91,2] = PR[GP1:90,2] + -1.172;
   1:L PR[91] R[100]mm/sec CNT100;
   1:  PR[GP1:91,1] = PR[GP1:90,1] + -58.738;
   1:  PR[GP1:91,2] = PR[GP1:90,2] + -12.300;
   1:L PR[91] R[100]mm/sec CNT100;
   1:  PR[GP1:91,1] = PR[GP1:90,1] + -58.467;
   1:  PR[GP1:91,2] = PR[GP1:90,2] + -13.221;
   1:L PR[91] R[100]mm/sec CNT100;
   1:  PR[GP1:91,1] = PR[GP1:90,1] + -58.024;
   1:  PR[GP1:91,2] = PR[GP1:90,2] + -14.088;
   1:L PR[91] R[100]mm/sec CNT100;
   1:  PR[GP1:91,1] = PR[GP1:90,1] + -51.838;
   1:  PR[GP1:91,2] = PR[GP1:90,2] + -24.381;
   1:L PR[91] R[100]mm/sec CNT100;
   1:  PR[GP1:91,1] = PR[GP1:90,1] + -51.439;
   1:  PR[GP1:91,2] = PR[GP1:90,2] + -24.900;
   1:L PR[91] R[100]mm/sec CNT100;
   1:  PR[GP1:91,1] = PR[GP1:90,1] + -50.984;
   1:  PR[GP1:91,2] = PR[GP1:90,2] + -25.309;
   1:L PR[91] R[100]mm/sec CNT100;
   1:  PR[GP1:91,1] = PR[GP1:90,1] + -40.836;
   1:  PR[GP1:91,2] = PR[GP1:90,2] + -33.487;
   1:L PR[91] R[100]mm/sec CNT100;
   1:  PR[GP1:91,1] = PR[GP1:90,1] + -40.700;
   1:  PR[GP1:91,2] = PR[GP1:90,2] + -33.572;
   1:L PR[91] R[100]mm/sec CNT100;
   1:  PR[GP1:91,1] = PR[GP1:90,1] + -40.554;
   1:  PR[GP1:91,2] = PR[GP1:90,2] + -33.631;
   1:L PR[91] R[100]mm/sec CNT100;
   1:  PR[GP1:91,1] = PR[GP1:90,1] + -35.313;
   1:  PR[GP1:91,2] = PR[GP1:90,2] + -35.480;
   1:L PR[91] R[100]mm/sec CNT100;
   1:  PR[GP1:91,1] = PR[GP1:90,1] + -27.955;
   1:  PR[GP1:91,2] = PR[GP1:90,2] + -38.192;
   1:L PR[91] R[100]mm/sec CNT100;
   1:  PR[GP1:91,1] = PR[GP1:90,1] + -27.336;
   1:  PR[GP1:91,2] = PR[GP1:90,2] + -38.396;
   1:L PR[91] R[100]mm/sec CNT100;
   1:  PR[GP1:91,1] = PR[GP1:90,1] + -14.768;
   1:  PR[GP1:91,2] = PR[GP1:90,2] + -38.619;
   1:L PR[91] R[100]mm/sec CNT100;
   1:  PR[GP1:91,1] = PR[GP1:90,1] + -12.784;
   1:  PR[GP1:91,2] = PR[GP1:90,2] + -38.539;
   1:L PR[91] R[100]mm/sec CNT100;
   1:  PR[GP1:91,1] = PR[GP1:90,1] + -5.746;
   1:  PR[GP1:91,2] = PR[GP1:90,2] + -36.346;
   1:L PR[91] R[100]mm/sec CNT100;
   1:  PR[GP1:91,1] = PR[GP1:90,1] + -1.997;
   1:  PR[GP1:91,2] = PR[GP1:90,2] + -35.122;
   1:L PR[91] R[100]mm/sec CNT100;
   1:  PR[GP1:91,1] = PR[GP1:90,1] + 2.206;
   1:  PR[GP1:91,2] = PR[GP1:90,2] + -35.131;
   1:L PR[91] R[100]mm/sec CNT100;
   1:  PR[GP1:91,1] = PR[GP1:90,1] + 5.953;
   1:  PR[GP1:91,2] = PR[GP1:90,2] + -36.343;
   1:L PR[91] R[100]mm/sec CNT100;
   1:  PR[GP1:91,1] = PR[GP1:90,1] + 13.035;
   1:  PR[GP1:91,2] = PR[GP1:90,2] + -38.549;
   1:L PR[91] R[100]mm/sec CNT100;
   1:  PR[GP1:91,1] = PR[GP1:90,1] + 14.977;
   1:  PR[GP1:91,2] = PR[GP1:90,2] + -38.618;
   1:L PR[91] R[100]mm/sec CNT100;
   1:  PR[GP1:91,1] = PR[GP1:90,1] + 27.546;
   1:  PR[GP1:91,2] = PR[GP1:90,2] + -38.396;
   1:L PR[91] R[100]mm/sec CNT100;
   1:  PR[GP1:91,1] = PR[GP1:90,1] + 28.166;
   1:  PR[GP1:91,2] = PR[GP1:90,2] + -38.193;
   1:L PR[91] R[100]mm/sec CNT100;
   1:  PR[GP1:91,1] = PR[GP1:90,1] + 35.525;
   1:  PR[GP1:91,2] = PR[GP1:90,2] + -35.482;
   1:L PR[91] R[100]mm/sec CNT100;
   1:  PR[GP1:91,1] = PR[GP1:90,1] + 40.922;
   1:  PR[GP1:91,2] = PR[GP1:90,2] + -33.569;
   1:L PR[91] R[100]mm/sec CNT100;
   1:  PR[GP1:91,1] = PR[GP1:90,1] + 41.034;
   1:  PR[GP1:91,2] = PR[GP1:90,2] + -33.500;
   1:L PR[91] R[100]mm/sec CNT100;
   1:  PR[GP1:91,1] = PR[GP1:90,1] + 41.207;
   1:  PR[GP1:91,2] = PR[GP1:90,2] + -33.346;
   1:L PR[91] R[100]mm/sec CNT100;
   1:  PR[GP1:91,1] = PR[GP1:90,1] + 51.652;
   1:  PR[GP1:91,2] = PR[GP1:90,2] + -24.892;
   1:L PR[91] R[100]mm/sec CNT100;
   1:  PR[GP1:91,1] = PR[GP1:90,1] + 52.035;
   1:  PR[GP1:91,2] = PR[GP1:90,2] + -24.394;
   1:L PR[91] R[100]mm/sec CNT100;
   1:  PR[GP1:91,1] = PR[GP1:90,1] + 52.395;
   1:  PR[GP1:91,2] = PR[GP1:90,2] + -23.704;
   1:L PR[91] R[100]mm/sec CNT100;
   1:  PR[GP1:91,1] = PR[GP1:90,1] + 58.682;
   1:  PR[GP1:91,2] = PR[GP1:90,2] + -13.229;
   1:L PR[91] R[100]mm/sec CNT100;
   1:  PR[GP1:91,1] = PR[GP1:90,1] + 58.939;
   1:  PR[GP1:91,2] = PR[GP1:90,2] + -12.370;
   1:L PR[91] R[100]mm/sec CNT100;
   1:  PR[GP1:91,1] = PR[GP1:90,1] + 59.036;
   1:  PR[GP1:91,2] = PR[GP1:90,2] + -11.326;
   1:L PR[91] R[100]mm/sec CNT100;
   1:  PR[GP1:91,1] = PR[GP1:90,1] + 61.114;
   1:  PR[GP1:91,2] = PR[GP1:90,2] + -0.045;
   1:L PR[91] R[100]mm/sec CNT100;
   1:  PR[GP1:91,1] = PR[GP1:90,1] + 61.012;
   1:  PR[GP1:91,2] = PR[GP1:90,2] + 1.060;
   1:L PR[91] R[100]mm/sec CNT100;
   1:  PR[GP1:91,1] = PR[GP1:90,1] + 58.948;
   1:  PR[GP1:91,2] = PR[GP1:90,2] + 12.196;
   1:L PR[91] R[100]mm/sec CNT100;
   1:  PR[GP1:91,1] = PR[GP1:90,1] + 58.678;
   1:  PR[GP1:91,2] = PR[GP1:90,2] + 13.100;
   1:L PR[91] R[100]mm/sec CNT100;
   1:  PR[GP1:91,1] = PR[GP1:90,1] + 58.234;
   1:  PR[GP1:91,2] = PR[GP1:90,2] + 13.961;
   1:L PR[91] R[100]mm/sec CNT100;
   1:  PR[GP1:91,1] = PR[GP1:90,1] + 52.052;
   1:  PR[GP1:91,2] = PR[GP1:90,2] + 24.230;
   1:L PR[91] R[100]mm/sec CNT100;
   1:  PR[GP1:91,1] = PR[GP1:90,1] + 51.648;
   1:  PR[GP1:91,2] = PR[GP1:90,2] + 24.754;
   1:L PR[91] R[100]mm/sec CNT100;
   1:  PR[GP1:91,1] = PR[GP1:90,1] + 51.195;
   1:  PR[GP1:91,2] = PR[GP1:90,2] + 25.159;
   1:L PR[91] R[100]mm/sec CNT100;
   1:  PR[GP1:91,1] = PR[GP1:90,1] + 41.057;
   1:  PR[GP1:91,2] = PR[GP1:90,2] + 33.342;
   1:L PR[91] R[100]mm/sec CNT100;
   1:  PR[GP1:91,1] = PR[GP1:90,1] + 40.933;
   1:  PR[GP1:91,2] = PR[GP1:90,2] + 33.419;
   1:L PR[91] R[100]mm/sec CNT100;
   1:  PR[GP1:91,1] = PR[GP1:90,1] + 35.525;
   1:  PR[GP1:91,2] = PR[GP1:90,2] + 35.338;
   1:L PR[91] R[100]mm/sec CNT100;
   1:  PR[GP1:91,1] = PR[GP1:90,1] + 28.181;
   1:  PR[GP1:91,2] = PR[GP1:90,2] + 38.046;
   1:L PR[91] R[100]mm/sec CNT100;
   1:  PR[GP1:91,1] = PR[GP1:90,1] + 27.563;
   1:  PR[GP1:91,2] = PR[GP1:90,2] + 38.249;
   1:L PR[91] R[100]mm/sec CNT100;
   1:  PR[GP1:91,1] = PR[GP1:90,1] + 14.994;
   1:  PR[GP1:91,2] = PR[GP1:90,2] + 38.477;
   1:L PR[91] R[100]mm/sec CNT100;
   1:  PR[GP1:91,1] = PR[GP1:90,1] + 13.053;
   1:  PR[GP1:91,2] = PR[GP1:90,2] + 38.407;
   1:L PR[91] R[100]mm/sec CNT100;
   1:  PR[GP1:91,1] = PR[GP1:90,1] + 7.227;
   1:  PR[GP1:91,2] = PR[GP1:90,2] + 36.607;
   1:L PR[91] R[100]mm/sec CNT100;
   1:  PR[GP1:91,1] = PR[GP1:90,1] + 2.206;
   1:  PR[GP1:91,2] = PR[GP1:90,2] + 34.986;
   1:L PR[91] R[100]mm/sec CNT100;
   1:  ! -- Layer/Ebene 124 -- !;
   1:  PR[91] = PR[90];
   1:  PR[GP1:91,1] = PR[GP1:90,1] + -1.971;
   1:  PR[GP1:91,2] = PR[GP1:90,2] + 35.164;
   1:  PR[GP1:91,3] = PR[GP1:90,3] + 75.945;
   1:L PR[91] R[100]mm/sec CNT100;
   1:  PR[GP1:91,1] = PR[GP1:90,1] + -5.750;
   1:  PR[GP1:91,2] = PR[GP1:90,2] + 36.397;
   1:L PR[91] R[100]mm/sec CNT100;
   1:  PR[GP1:91,1] = PR[GP1:90,1] + -12.545;
   1:  PR[GP1:91,2] = PR[GP1:90,2] + 38.497;
   1:L PR[91] R[100]mm/sec CNT100;
   1:  PR[GP1:91,1] = PR[GP1:90,1] + -14.822;
   1:  PR[GP1:91,2] = PR[GP1:90,2] + 38.578;
   1:L PR[91] R[100]mm/sec CNT100;
   1:  PR[GP1:91,1] = PR[GP1:90,1] + -27.091;
   1:  PR[GP1:91,2] = PR[GP1:90,2] + 38.355;
   1:L PR[91] R[100]mm/sec CNT100;
   1:  PR[GP1:91,1] = PR[GP1:90,1] + -28.039;
   1:  PR[GP1:91,2] = PR[GP1:90,2] + 38.044;
   1:L PR[91] R[100]mm/sec CNT100;
   1:  PR[GP1:91,1] = PR[GP1:90,1] + -38.773;
   1:  PR[GP1:91,2] = PR[GP1:90,2] + 34.082;
   1:L PR[91] R[100]mm/sec CNT100;
   1:  PR[GP1:91,1] = PR[GP1:90,1] + -40.532;
   1:  PR[GP1:91,2] = PR[GP1:90,2] + 33.458;
   1:L PR[91] R[100]mm/sec CNT100;
   1:  PR[GP1:91,1] = PR[GP1:90,1] + -51.270;
   1:  PR[GP1:91,2] = PR[GP1:90,2] + 24.762;
   1:L PR[91] R[100]mm/sec CNT100;
   1:  PR[GP1:91,1] = PR[GP1:90,1] + -51.547;
   1:  PR[GP1:91,2] = PR[GP1:90,2] + 24.402;
   1:L PR[91] R[100]mm/sec CNT100;
   1:  PR[GP1:91,1] = PR[GP1:90,1] + -51.822;
   1:  PR[GP1:91,2] = PR[GP1:90,2] + 23.868;
   1:L PR[91] R[100]mm/sec CNT100;
   1:  PR[GP1:91,1] = PR[GP1:90,1] + -58.287;
   1:  PR[GP1:91,2] = PR[GP1:90,2] + 13.069;
   1:L PR[91] R[100]mm/sec CNT100;
   1:  PR[GP1:91,1] = PR[GP1:90,1] + -58.499;
   1:  PR[GP1:91,2] = PR[GP1:90,2] + 12.351;
   1:L PR[91] R[100]mm/sec CNT100;
   1:  PR[GP1:91,1] = PR[GP1:90,1] + -58.577;
   1:  PR[GP1:91,2] = PR[GP1:90,2] + 11.498;
   1:L PR[91] R[100]mm/sec CNT100;
   1:  PR[GP1:91,1] = PR[GP1:90,1] + -60.714;
   1:  PR[GP1:91,2] = PR[GP1:90,2] + -0.100;
   1:L PR[91] R[100]mm/sec CNT100;
   1:  PR[GP1:91,1] = PR[GP1:90,1] + -60.632;
   1:  PR[GP1:91,2] = PR[GP1:90,2] + -1.015;
   1:L PR[91] R[100]mm/sec CNT100;
   1:  PR[GP1:91,1] = PR[GP1:90,1] + -58.505;
   1:  PR[GP1:91,2] = PR[GP1:90,2] + -12.472;
   1:L PR[91] R[100]mm/sec CNT100;
   1:  PR[GP1:91,1] = PR[GP1:90,1] + -58.280;
   1:  PR[GP1:91,2] = PR[GP1:90,2] + -13.236;
   1:L PR[91] R[100]mm/sec CNT100;
   1:  PR[GP1:91,1] = PR[GP1:90,1] + -57.911;
   1:  PR[GP1:91,2] = PR[GP1:90,2] + -13.959;
   1:L PR[91] R[100]mm/sec CNT100;
   1:  PR[GP1:91,1] = PR[GP1:90,1] + -51.553;
   1:  PR[GP1:91,2] = PR[GP1:90,2] + -24.537;
   1:L PR[91] R[100]mm/sec CNT100;
   1:  PR[GP1:91,1] = PR[GP1:90,1] + -51.255;
   1:  PR[GP1:91,2] = PR[GP1:90,2] + -24.925;
   1:L PR[91] R[100]mm/sec CNT100;
   1:  PR[GP1:91,1] = PR[GP1:90,1] + -50.913;
   1:  PR[GP1:91,2] = PR[GP1:90,2] + -25.232;
   1:L PR[91] R[100]mm/sec CNT100;
   1:  PR[GP1:91,1] = PR[GP1:90,1] + -40.530;
   1:  PR[GP1:91,2] = PR[GP1:90,2] + -33.600;
   1:L PR[91] R[100]mm/sec CNT100;
   1:  PR[GP1:91,1] = PR[GP1:90,1] + -40.482;
   1:  PR[GP1:91,2] = PR[GP1:90,2] + -33.625;
   1:L PR[91] R[100]mm/sec CNT100;
   1:  PR[GP1:91,1] = PR[GP1:90,1] + -38.774;
   1:  PR[GP1:91,2] = PR[GP1:90,2] + -34.227;
   1:L PR[91] R[100]mm/sec CNT100;
   1:  PR[GP1:91,1] = PR[GP1:90,1] + -28.024;
   1:  PR[GP1:91,2] = PR[GP1:90,2] + -38.190;
   1:L PR[91] R[100]mm/sec CNT100;
   1:  PR[GP1:91,1] = PR[GP1:90,1] + -27.075;
   1:  PR[GP1:91,2] = PR[GP1:90,2] + -38.502;
   1:L PR[91] R[100]mm/sec CNT100;
   1:  PR[GP1:91,1] = PR[GP1:90,1] + -14.805;
   1:  PR[GP1:91,2] = PR[GP1:90,2] + -38.719;
   1:L PR[91] R[100]mm/sec CNT100;
   1:  PR[GP1:91,1] = PR[GP1:90,1] + -12.528;
   1:  PR[GP1:91,2] = PR[GP1:90,2] + -38.638;
   1:L PR[91] R[100]mm/sec CNT100;
   1:  PR[GP1:91,1] = PR[GP1:90,1] + -4.271;
   1:  PR[GP1:91,2] = PR[GP1:90,2] + -36.067;
   1:L PR[91] R[100]mm/sec CNT100;
   1:  PR[GP1:91,1] = PR[GP1:90,1] + -1.971;
   1:  PR[GP1:91,2] = PR[GP1:90,2] + -35.317;
   1:L PR[91] R[100]mm/sec CNT100;
   1:  PR[GP1:91,1] = PR[GP1:90,1] + 2.179;
   1:  PR[GP1:91,2] = PR[GP1:90,2] + -35.322;
   1:L PR[91] R[100]mm/sec CNT100;
   1:  PR[GP1:91,1] = PR[GP1:90,1] + 4.478;
   1:  PR[GP1:91,2] = PR[GP1:90,2] + -36.065;
   1:L PR[91] R[100]mm/sec CNT100;
   1:  PR[GP1:91,1] = PR[GP1:90,1] + 12.738;
   1:  PR[GP1:91,2] = PR[GP1:90,2] + -38.637;
   1:L PR[91] R[100]mm/sec CNT100;
   1:  PR[GP1:91,1] = PR[GP1:90,1] + 15.016;
   1:  PR[GP1:91,2] = PR[GP1:90,2] + -38.719;
   1:L PR[91] R[100]mm/sec CNT100;
   1:  PR[GP1:91,1] = PR[GP1:90,1] + 27.286;
   1:  PR[GP1:91,2] = PR[GP1:90,2] + -38.502;
   1:L PR[91] R[100]mm/sec CNT100;
   1:  PR[GP1:91,1] = PR[GP1:90,1] + 28.235;
   1:  PR[GP1:91,2] = PR[GP1:90,2] + -38.191;
   1:L PR[91] R[100]mm/sec CNT100;
   1:  PR[GP1:91,1] = PR[GP1:90,1] + 38.986;
   1:  PR[GP1:91,2] = PR[GP1:90,2] + -34.230;
   1:L PR[91] R[100]mm/sec CNT100;
   1:  PR[GP1:91,1] = PR[GP1:90,1] + 40.732;
   1:  PR[GP1:91,2] = PR[GP1:90,2] + -33.612;
   1:L PR[91] R[100]mm/sec CNT100;
   1:  PR[GP1:91,1] = PR[GP1:90,1] + 51.471;
   1:  PR[GP1:91,2] = PR[GP1:90,2] + -24.914;
   1:L PR[91] R[100]mm/sec CNT100;
   1:  PR[GP1:91,1] = PR[GP1:90,1] + 51.751;
   1:  PR[GP1:91,2] = PR[GP1:90,2] + -24.549;
   1:L PR[91] R[100]mm/sec CNT100;
   1:  PR[GP1:91,1] = PR[GP1:90,1] + 52.027;
   1:  PR[GP1:91,2] = PR[GP1:90,2] + -24.020;
   1:L PR[91] R[100]mm/sec CNT100;
   1:  PR[GP1:91,1] = PR[GP1:90,1] + 58.496;
   1:  PR[GP1:91,2] = PR[GP1:90,2] + -13.243;
   1:L PR[91] R[100]mm/sec CNT100;
   1:  PR[GP1:91,1] = PR[GP1:90,1] + 58.707;
   1:  PR[GP1:91,2] = PR[GP1:90,2] + -12.537;
   1:L PR[91] R[100]mm/sec CNT100;
   1:  PR[GP1:91,1] = PR[GP1:90,1] + 58.788;
   1:  PR[GP1:91,2] = PR[GP1:90,2] + -11.661;
   1:L PR[91] R[100]mm/sec CNT100;
   1:  PR[GP1:91,1] = PR[GP1:90,1] + 60.928;
   1:  PR[GP1:91,2] = PR[GP1:90,2] + -0.045;
   1:L PR[91] R[100]mm/sec CNT100;
   1:  PR[GP1:91,1] = PR[GP1:90,1] + 60.841;
   1:  PR[GP1:91,2] = PR[GP1:90,2] + 0.899;
   1:L PR[91] R[100]mm/sec CNT100;
   1:  PR[GP1:91,1] = PR[GP1:90,1] + 58.716;
   1:  PR[GP1:91,2] = PR[GP1:90,2] + 12.364;
   1:L PR[91] R[100]mm/sec CNT100;
   1:  PR[GP1:91,1] = PR[GP1:90,1] + 58.491;
   1:  PR[GP1:91,2] = PR[GP1:90,2] + 13.114;
   1:L PR[91] R[100]mm/sec CNT100;
   1:  PR[GP1:91,1] = PR[GP1:90,1] + 58.122;
   1:  PR[GP1:91,2] = PR[GP1:90,2] + 13.831;
   1:L PR[91] R[100]mm/sec CNT100;
   1:  PR[GP1:91,1] = PR[GP1:90,1] + 51.768;
   1:  PR[GP1:91,2] = PR[GP1:90,2] + 24.385;
   1:L PR[91] R[100]mm/sec CNT100;
   1:  PR[GP1:91,1] = PR[GP1:90,1] + 51.467;
   1:  PR[GP1:91,2] = PR[GP1:90,2] + 24.776;
   1:L PR[91] R[100]mm/sec CNT100;
   1:  PR[GP1:91,1] = PR[GP1:90,1] + 51.126;
   1:  PR[GP1:91,2] = PR[GP1:90,2] + 25.080;
   1:L PR[91] R[100]mm/sec CNT100;
   1:  PR[GP1:91,1] = PR[GP1:90,1] + 40.743;
   1:  PR[GP1:91,2] = PR[GP1:90,2] + 33.461;
   1:L PR[91] R[100]mm/sec CNT100;
   1:  PR[GP1:91,1] = PR[GP1:90,1] + 38.986;
   1:  PR[GP1:91,2] = PR[GP1:90,2] + 34.085;
   1:L PR[91] R[100]mm/sec CNT100;
   1:  PR[GP1:91,1] = PR[GP1:90,1] + 28.250;
   1:  PR[GP1:91,2] = PR[GP1:90,2] + 38.044;
   1:L PR[91] R[100]mm/sec CNT100;
   1:  PR[GP1:91,1] = PR[GP1:90,1] + 27.302;
   1:  PR[GP1:91,2] = PR[GP1:90,2] + 38.355;
   1:L PR[91] R[100]mm/sec CNT100;
   1:  PR[GP1:91,1] = PR[GP1:90,1] + 15.032;
   1:  PR[GP1:91,2] = PR[GP1:90,2] + 38.578;
   1:L PR[91] R[100]mm/sec CNT100;
   1:  PR[GP1:91,1] = PR[GP1:90,1] + 12.755;
   1:  PR[GP1:91,2] = PR[GP1:90,2] + 38.496;
   1:L PR[91] R[100]mm/sec CNT100;
   1:  PR[GP1:91,1] = PR[GP1:90,1] + 5.957;
   1:  PR[GP1:91,2] = PR[GP1:90,2] + 36.395;
   1:L PR[91] R[100]mm/sec CNT100;
   1:  PR[GP1:91,1] = PR[GP1:90,1] + 2.180;
   1:  PR[GP1:91,2] = PR[GP1:90,2] + 35.175;
   1:L PR[91] R[100]mm/sec CNT100;
   1:  ! -- Layer/Ebene 125 -- !;
   1:  PR[91] = PR[90];
   1:  PR[GP1:91,1] = PR[GP1:90,1] + -1.944;
   1:  PR[GP1:91,2] = PR[GP1:90,2] + 35.358;
   1:  PR[GP1:91,3] = PR[GP1:90,3] + 76.555;
   1:L PR[91] R[100]mm/sec CNT100;
   1:  PR[GP1:91,1] = PR[GP1:90,1] + -4.480;
   1:  PR[GP1:91,2] = PR[GP1:90,2] + 36.185;
   1:L PR[91] R[100]mm/sec CNT100;
   1:  PR[GP1:91,1] = PR[GP1:90,1] + -12.247;
   1:  PR[GP1:91,2] = PR[GP1:90,2] + 38.585;
   1:L PR[91] R[100]mm/sec CNT100;
   1:  PR[GP1:91,1] = PR[GP1:90,1] + -14.860;
   1:  PR[GP1:91,2] = PR[GP1:90,2] + 38.679;
   1:L PR[91] R[100]mm/sec CNT100;
   1:  PR[GP1:91,1] = PR[GP1:90,1] + -26.830;
   1:  PR[GP1:91,2] = PR[GP1:90,2] + 38.461;
   1:L PR[91] R[100]mm/sec CNT100;
   1:  PR[GP1:91,1] = PR[GP1:90,1] + -28.107;
   1:  PR[GP1:91,2] = PR[GP1:90,2] + 38.042;
   1:L PR[91] R[100]mm/sec CNT100;
   1:  PR[GP1:91,1] = PR[GP1:90,1] + -40.295;
   1:  PR[GP1:91,2] = PR[GP1:90,2] + 33.544;
   1:L PR[91] R[100]mm/sec CNT100;
   1:  PR[GP1:91,1] = PR[GP1:90,1] + -42.063;
   1:  PR[GP1:91,2] = PR[GP1:90,2] + 32.090;
   1:L PR[91] R[100]mm/sec CNT100;
   1:  PR[GP1:91,1] = PR[GP1:90,1] + -51.087;
   1:  PR[GP1:91,2] = PR[GP1:90,2] + 24.787;
   1:L PR[91] R[100]mm/sec CNT100;
   1:  PR[GP1:91,1] = PR[GP1:90,1] + -51.262;
   1:  PR[GP1:91,2] = PR[GP1:90,2] + 24.558;
   1:L PR[91] R[100]mm/sec CNT100;
   1:  PR[GP1:91,1] = PR[GP1:90,1] + -51.454;
   1:  PR[GP1:91,2] = PR[GP1:90,2] + 24.186;
   1:L PR[91] R[100]mm/sec CNT100;
   1:  PR[GP1:91,1] = PR[GP1:90,1] + -58.100;
   1:  PR[GP1:91,2] = PR[GP1:90,2] + 13.085;
   1:L PR[91] R[100]mm/sec CNT100;
   1:  PR[GP1:91,1] = PR[GP1:90,1] + -58.266;
   1:  PR[GP1:91,2] = PR[GP1:90,2] + 12.523;
   1:L PR[91] R[100]mm/sec CNT100;
   1:  PR[GP1:91,1] = PR[GP1:90,1] + -58.329;
   1:  PR[GP1:91,2] = PR[GP1:90,2] + 11.833;
   1:L PR[91] R[100]mm/sec CNT100;
   1:  PR[GP1:91,1] = PR[GP1:90,1] + -60.528;
   1:  PR[GP1:91,2] = PR[GP1:90,2] + -0.100;
   1:L PR[91] R[100]mm/sec CNT100;
   1:  PR[GP1:91,1] = PR[GP1:90,1] + -60.460;
   1:  PR[GP1:91,2] = PR[GP1:90,2] + -0.859;
   1:L PR[91] R[100]mm/sec CNT100;
   1:  PR[GP1:91,1] = PR[GP1:90,1] + -58.272;
   1:  PR[GP1:91,2] = PR[GP1:90,2] + -12.644;
   1:L PR[91] R[100]mm/sec CNT100;
   1:  PR[GP1:91,1] = PR[GP1:90,1] + -58.093;
   1:  PR[GP1:91,2] = PR[GP1:90,2] + -13.252;
   1:L PR[91] R[100]mm/sec CNT100;
   1:  PR[GP1:91,1] = PR[GP1:90,1] + -57.798;
   1:  PR[GP1:91,2] = PR[GP1:90,2] + -13.829;
   1:L PR[91] R[100]mm/sec CNT100;
   1:  PR[GP1:91,1] = PR[GP1:90,1] + -51.269;
   1:  PR[GP1:91,2] = PR[GP1:90,2] + -24.693;
   1:L PR[91] R[100]mm/sec CNT100;
   1:  PR[GP1:91,1] = PR[GP1:90,1] + -51.072;
   1:  PR[GP1:91,2] = PR[GP1:90,2] + -24.949;
   1:L PR[91] R[100]mm/sec CNT100;
   1:  PR[GP1:91,1] = PR[GP1:90,1] + -50.843;
   1:  PR[GP1:91,2] = PR[GP1:90,2] + -25.154;
   1:L PR[91] R[100]mm/sec CNT100;
   1:  PR[GP1:91,1] = PR[GP1:90,1] + -42.063;
   1:  PR[GP1:91,2] = PR[GP1:90,2] + -32.231;
   1:L PR[91] R[100]mm/sec CNT100;
   1:  PR[GP1:91,1] = PR[GP1:90,1] + -40.284;
   1:  PR[GP1:91,2] = PR[GP1:90,2] + -33.694;
   1:L PR[91] R[100]mm/sec CNT100;
   1:  PR[GP1:91,1] = PR[GP1:90,1] + -28.093;
   1:  PR[GP1:91,2] = PR[GP1:90,2] + -38.188;
   1:L PR[91] R[100]mm/sec CNT100;
   1:  PR[GP1:91,1] = PR[GP1:90,1] + -26.814;
   1:  PR[GP1:91,2] = PR[GP1:90,2] + -38.608;
   1:L PR[91] R[100]mm/sec CNT100;
   1:  PR[GP1:91,1] = PR[GP1:90,1] + -14.844;
   1:  PR[GP1:91,2] = PR[GP1:90,2] + -38.820;
   1:L PR[91] R[100]mm/sec CNT100;
   1:  PR[GP1:91,1] = PR[GP1:90,1] + -12.231;
   1:  PR[GP1:91,2] = PR[GP1:90,2] + -38.727;
   1:L PR[91] R[100]mm/sec CNT100;
   1:  PR[GP1:91,1] = PR[GP1:90,1] + -2.796;
   1:  PR[GP1:91,2] = PR[GP1:90,2] + -35.789;
   1:L PR[91] R[100]mm/sec CNT100;
   1:  PR[GP1:91,1] = PR[GP1:90,1] + -1.944;
   1:  PR[GP1:91,2] = PR[GP1:90,2] + -35.511;
   1:L PR[91] R[100]mm/sec CNT100;
   1:  PR[GP1:91,1] = PR[GP1:90,1] + 2.150;
   1:  PR[GP1:91,2] = PR[GP1:90,2] + -35.512;
   1:L PR[91] R[100]mm/sec CNT100;
   1:  PR[GP1:91,1] = PR[GP1:90,1] + 12.442;
   1:  PR[GP1:91,2] = PR[GP1:90,2] + -38.726;
   1:L PR[91] R[100]mm/sec CNT100;
   1:  PR[GP1:91,1] = PR[GP1:90,1] + 15.055;
   1:  PR[GP1:91,2] = PR[GP1:90,2] + -38.819;
   1:L PR[91] R[100]mm/sec CNT100;
   1:  PR[GP1:91,1] = PR[GP1:90,1] + 27.025;
   1:  PR[GP1:91,2] = PR[GP1:90,2] + -38.608;
   1:L PR[91] R[100]mm/sec CNT100;
   1:  PR[GP1:91,1] = PR[GP1:90,1] + 28.304;
   1:  PR[GP1:91,2] = PR[GP1:90,2] + -38.189;
   1:L PR[91] R[100]mm/sec CNT100;
   1:  PR[GP1:91,1] = PR[GP1:90,1] + 40.495;
   1:  PR[GP1:91,2] = PR[GP1:90,2] + -33.698;
   1:L PR[91] R[100]mm/sec CNT100;
   1:  PR[GP1:91,1] = PR[GP1:90,1] + 42.275;
   1:  PR[GP1:91,2] = PR[GP1:90,2] + -32.233;
   1:L PR[91] R[100]mm/sec CNT100;
   1:  PR[GP1:91,1] = PR[GP1:90,1] + 51.289;
   1:  PR[GP1:91,2] = PR[GP1:90,2] + -24.936;
   1:L PR[91] R[100]mm/sec CNT100;
   1:  PR[GP1:91,1] = PR[GP1:90,1] + 51.468;
   1:  PR[GP1:91,2] = PR[GP1:90,2] + -24.704;
   1:L PR[91] R[100]mm/sec CNT100;
   1:  PR[GP1:91,1] = PR[GP1:90,1] + 51.660;
   1:  PR[GP1:91,2] = PR[GP1:90,2] + -24.335;
   1:L PR[91] R[100]mm/sec CNT100;
   1:  PR[GP1:91,1] = PR[GP1:90,1] + 58.309;
   1:  PR[GP1:91,2] = PR[GP1:90,2] + -13.257;
   1:L PR[91] R[100]mm/sec CNT100;
   1:  PR[GP1:91,1] = PR[GP1:90,1] + 58.474;
   1:  PR[GP1:91,2] = PR[GP1:90,2] + -12.705;
   1:L PR[91] R[100]mm/sec CNT100;
   1:  PR[GP1:91,1] = PR[GP1:90,1] + 58.540;
   1:  PR[GP1:91,2] = PR[GP1:90,2] + -11.996;
   1:L PR[91] R[100]mm/sec CNT100;
   1:  PR[GP1:91,1] = PR[GP1:90,1] + 60.741;
   1:  PR[GP1:91,2] = PR[GP1:90,2] + -0.045;
   1:L PR[91] R[100]mm/sec CNT100;
   1:  PR[GP1:91,1] = PR[GP1:90,1] + 60.669;
   1:  PR[GP1:91,2] = PR[GP1:90,2] + 0.738;
   1:L PR[91] R[100]mm/sec CNT100;
   1:  PR[GP1:91,1] = PR[GP1:90,1] + 58.483;
   1:  PR[GP1:91,2] = PR[GP1:90,2] + 12.531;
   1:L PR[91] R[100]mm/sec CNT100;
   1:  PR[GP1:91,1] = PR[GP1:90,1] + 58.305;
   1:  PR[GP1:91,2] = PR[GP1:90,2] + 13.128;
   1:L PR[91] R[100]mm/sec CNT100;
   1:  PR[GP1:91,1] = PR[GP1:90,1] + 58.010;
   1:  PR[GP1:91,2] = PR[GP1:90,2] + 13.700;
   1:L PR[91] R[100]mm/sec CNT100;
   1:  PR[GP1:91,1] = PR[GP1:90,1] + 51.484;
   1:  PR[GP1:91,2] = PR[GP1:90,2] + 24.539;
   1:L PR[91] R[100]mm/sec CNT100;
   1:  PR[GP1:91,1] = PR[GP1:90,1] + 51.285;
   1:  PR[GP1:91,2] = PR[GP1:90,2] + 24.798;
   1:L PR[91] R[100]mm/sec CNT100;
   1:  PR[GP1:91,1] = PR[GP1:90,1] + 51.058;
   1:  PR[GP1:91,2] = PR[GP1:90,2] + 25.001;
   1:L PR[91] R[100]mm/sec CNT100;
   1:  PR[GP1:91,1] = PR[GP1:90,1] + 42.276;
   1:  PR[GP1:91,2] = PR[GP1:90,2] + 32.090;
   1:L PR[91] R[100]mm/sec CNT100;
   1:  PR[GP1:91,1] = PR[GP1:90,1] + 40.506;
   1:  PR[GP1:91,2] = PR[GP1:90,2] + 33.547;
   1:L PR[91] R[100]mm/sec CNT100;
   1:  PR[GP1:91,1] = PR[GP1:90,1] + 28.318;
   1:  PR[GP1:91,2] = PR[GP1:90,2] + 38.042;
   1:L PR[91] R[100]mm/sec CNT100;
   1:  PR[GP1:91,1] = PR[GP1:90,1] + 27.040;
   1:  PR[GP1:91,2] = PR[GP1:90,2] + 38.461;
   1:L PR[91] R[100]mm/sec CNT100;
   1:  PR[GP1:91,1] = PR[GP1:90,1] + 15.071;
   1:  PR[GP1:91,2] = PR[GP1:90,2] + 38.678;
   1:L PR[91] R[100]mm/sec CNT100;
   1:  PR[GP1:91,1] = PR[GP1:90,1] + 12.458;
   1:  PR[GP1:91,2] = PR[GP1:90,2] + 38.585;
   1:L PR[91] R[100]mm/sec CNT100;
   1:  PR[GP1:91,1] = PR[GP1:90,1] + 4.687;
   1:  PR[GP1:91,2] = PR[GP1:90,2] + 36.183;
   1:L PR[91] R[100]mm/sec CNT100;
   1:  PR[GP1:91,1] = PR[GP1:90,1] + 2.153;
   1:  PR[GP1:91,2] = PR[GP1:90,2] + 35.365;
   1:L PR[91] R[100]mm/sec CNT100;
   1:  ! -- Layer/Ebene 126 -- !;
   1:  PR[91] = PR[90];
   1:  PR[GP1:91,1] = PR[GP1:90,1] + -1.917;
   1:  PR[GP1:91,2] = PR[GP1:90,2] + 35.552;
   1:  PR[GP1:91,3] = PR[GP1:90,3] + 77.165;
   1:L PR[91] R[100]mm/sec CNT100;
   1:  PR[GP1:91,1] = PR[GP1:90,1] + -3.210;
   1:  PR[GP1:91,2] = PR[GP1:90,2] + 35.973;
   1:L PR[91] R[100]mm/sec CNT100;
   1:  PR[GP1:91,1] = PR[GP1:90,1] + -11.950;
   1:  PR[GP1:91,2] = PR[GP1:90,2] + 38.674;
   1:L PR[91] R[100]mm/sec CNT100;
   1:  PR[GP1:91,1] = PR[GP1:90,1] + -14.899;
   1:  PR[GP1:91,2] = PR[GP1:90,2] + 38.780;
   1:L PR[91] R[100]mm/sec CNT100;
   1:  PR[GP1:91,1] = PR[GP1:90,1] + -26.568;
   1:  PR[GP1:91,2] = PR[GP1:90,2] + 38.567;
   1:L PR[91] R[100]mm/sec CNT100;
   1:  PR[GP1:91,1] = PR[GP1:90,1] + -28.176;
   1:  PR[GP1:91,2] = PR[GP1:90,2] + 38.040;
   1:L PR[91] R[100]mm/sec CNT100;
   1:  PR[GP1:91,1] = PR[GP1:90,1] + -40.079;
   1:  PR[GP1:91,2] = PR[GP1:90,2] + 33.647;
   1:L PR[91] R[100]mm/sec CNT100;
   1:  PR[GP1:91,1] = PR[GP1:90,1] + -40.421;
   1:  PR[GP1:91,2] = PR[GP1:90,2] + 33.376;
   1:L PR[91] R[100]mm/sec CNT100;
   1:  PR[GP1:91,1] = PR[GP1:90,1] + -45.530;
   1:  PR[GP1:91,2] = PR[GP1:90,2] + 29.159;
   1:L PR[91] R[100]mm/sec CNT100;
   1:  PR[GP1:91,1] = PR[GP1:90,1] + -50.903;
   1:  PR[GP1:91,2] = PR[GP1:90,2] + 24.811;
   1:L PR[91] R[100]mm/sec CNT100;
   1:  PR[GP1:91,1] = PR[GP1:90,1] + -50.978;
   1:  PR[GP1:91,2] = PR[GP1:90,2] + 24.714;
   1:L PR[91] R[100]mm/sec CNT100;
   1:  PR[GP1:91,1] = PR[GP1:90,1] + -51.086;
   1:  PR[GP1:91,2] = PR[GP1:90,2] + 24.504;
   1:L PR[91] R[100]mm/sec CNT100;
   1:  PR[GP1:91,1] = PR[GP1:90,1] + -57.913;
   1:  PR[GP1:91,2] = PR[GP1:90,2] + 13.100;
   1:L PR[91] R[100]mm/sec CNT100;
   1:  PR[GP1:91,1] = PR[GP1:90,1] + -58.032;
   1:  PR[GP1:91,2] = PR[GP1:90,2] + 12.694;
   1:L PR[91] R[100]mm/sec CNT100;
   1:  PR[GP1:91,1] = PR[GP1:90,1] + -58.081;
   1:  PR[GP1:91,2] = PR[GP1:90,2] + 12.167;
   1:L PR[91] R[100]mm/sec CNT100;
   1:  PR[GP1:91,1] = PR[GP1:90,1] + -60.342;
   1:  PR[GP1:91,2] = PR[GP1:90,2] + -0.100;
   1:L PR[91] R[100]mm/sec CNT100;
   1:  PR[GP1:91,1] = PR[GP1:90,1] + -60.287;
   1:  PR[GP1:91,2] = PR[GP1:90,2] + -0.703;
   1:L PR[91] R[100]mm/sec CNT100;
   1:  PR[GP1:91,1] = PR[GP1:90,1] + -58.039;
   1:  PR[GP1:91,2] = PR[GP1:90,2] + -12.815;
   1:L PR[91] R[100]mm/sec CNT100;
   1:  PR[GP1:91,1] = PR[GP1:90,1] + -57.906;
   1:  PR[GP1:91,2] = PR[GP1:90,2] + -13.268;
   1:L PR[91] R[100]mm/sec CNT100;
   1:  PR[GP1:91,1] = PR[GP1:90,1] + -57.686;
   1:  PR[GP1:91,2] = PR[GP1:90,2] + -13.699;
   1:L PR[91] R[100]mm/sec CNT100;
   1:  PR[GP1:91,1] = PR[GP1:90,1] + -50.984;
   1:  PR[GP1:91,2] = PR[GP1:90,2] + -24.849;
   1:L PR[91] R[100]mm/sec CNT100;
   1:  PR[GP1:91,1] = PR[GP1:90,1] + -50.888;
   1:  PR[GP1:91,2] = PR[GP1:90,2] + -24.974;
   1:L PR[91] R[100]mm/sec CNT100;
   1:  PR[GP1:91,1] = PR[GP1:90,1] + -50.773;
   1:  PR[GP1:91,2] = PR[GP1:90,2] + -25.077;
   1:L PR[91] R[100]mm/sec CNT100;
   1:  PR[GP1:91,1] = PR[GP1:90,1] + -45.531;
   1:  PR[GP1:91,2] = PR[GP1:90,2] + -29.302;
   1:L PR[91] R[100]mm/sec CNT100;
   1:  PR[GP1:91,1] = PR[GP1:90,1] + -40.411;
   1:  PR[GP1:91,2] = PR[GP1:90,2] + -33.526;
   1:L PR[91] R[100]mm/sec CNT100;
   1:  PR[GP1:91,1] = PR[GP1:90,1] + -40.068;
   1:  PR[GP1:91,2] = PR[GP1:90,2] + -33.797;
   1:L PR[91] R[100]mm/sec CNT100;
   1:  PR[GP1:91,1] = PR[GP1:90,1] + -28.162;
   1:  PR[GP1:91,2] = PR[GP1:90,2] + -38.186;
   1:L PR[91] R[100]mm/sec CNT100;
   1:  PR[GP1:91,1] = PR[GP1:90,1] + -26.553;
   1:  PR[GP1:91,2] = PR[GP1:90,2] + -38.714;
   1:L PR[91] R[100]mm/sec CNT100;
   1:  PR[GP1:91,1] = PR[GP1:90,1] + -14.882;
   1:  PR[GP1:91,2] = PR[GP1:90,2] + -38.921;
   1:L PR[91] R[100]mm/sec CNT100;
   1:  PR[GP1:91,1] = PR[GP1:90,1] + -11.934;
   1:  PR[GP1:91,2] = PR[GP1:90,2] + -38.816;
   1:L PR[91] R[100]mm/sec CNT100;
   1:  PR[GP1:91,1] = PR[GP1:90,1] + -1.913;
   1:  PR[GP1:91,2] = PR[GP1:90,2] + -35.696;
   1:L PR[91] R[100]mm/sec CNT100;
   1:  PR[GP1:91,1] = PR[GP1:90,1] + 2.123;
   1:  PR[GP1:91,2] = PR[GP1:90,2] + -35.695;
   1:L PR[91] R[100]mm/sec CNT100;
   1:  PR[GP1:91,1] = PR[GP1:90,1] + 12.145;
   1:  PR[GP1:91,2] = PR[GP1:90,2] + -38.815;
   1:L PR[91] R[100]mm/sec CNT100;
   1:  PR[GP1:91,1] = PR[GP1:90,1] + 15.093;
   1:  PR[GP1:91,2] = PR[GP1:90,2] + -38.920;
   1:L PR[91] R[100]mm/sec CNT100;
   1:  PR[GP1:91,1] = PR[GP1:90,1] + 26.764;
   1:  PR[GP1:91,2] = PR[GP1:90,2] + -38.714;
   1:L PR[91] R[100]mm/sec CNT100;
   1:  PR[GP1:91,1] = PR[GP1:90,1] + 28.373;
   1:  PR[GP1:91,2] = PR[GP1:90,2] + -38.187;
   1:L PR[91] R[100]mm/sec CNT100;
   1:  PR[GP1:91,1] = PR[GP1:90,1] + 40.279;
   1:  PR[GP1:91,2] = PR[GP1:90,2] + -33.801;
   1:L PR[91] R[100]mm/sec CNT100;
   1:  PR[GP1:91,1] = PR[GP1:90,1] + 40.623;
   1:  PR[GP1:91,2] = PR[GP1:90,2] + -33.529;
   1:L PR[91] R[100]mm/sec CNT100;
   1:  PR[GP1:91,1] = PR[GP1:90,1] + 45.743;
   1:  PR[GP1:91,2] = PR[GP1:90,2] + -29.301;
   1:L PR[91] R[100]mm/sec CNT100;
   1:  PR[GP1:91,1] = PR[GP1:90,1] + 51.108;
   1:  PR[GP1:91,2] = PR[GP1:90,2] + -24.958;
   1:L PR[91] R[100]mm/sec CNT100;
   1:  PR[GP1:91,1] = PR[GP1:90,1] + 51.184;
   1:  PR[GP1:91,2] = PR[GP1:90,2] + -24.859;
   1:L PR[91] R[100]mm/sec CNT100;
   1:  PR[GP1:91,1] = PR[GP1:90,1] + 51.292;
   1:  PR[GP1:91,2] = PR[GP1:90,2] + -24.651;
   1:L PR[91] R[100]mm/sec CNT100;
   1:  PR[GP1:91,1] = PR[GP1:90,1] + 58.123;
   1:  PR[GP1:91,2] = PR[GP1:90,2] + -13.271;
   1:L PR[91] R[100]mm/sec CNT100;
   1:  PR[GP1:91,1] = PR[GP1:90,1] + 58.242;
   1:  PR[GP1:91,2] = PR[GP1:90,2] + -12.873;
   1:L PR[91] R[100]mm/sec CNT100;
   1:  PR[GP1:91,1] = PR[GP1:90,1] + 58.292;
   1:  PR[GP1:91,2] = PR[GP1:90,2] + -12.331;
   1:L PR[91] R[100]mm/sec CNT100;
   1:  PR[GP1:91,1] = PR[GP1:90,1] + 60.555;
   1:  PR[GP1:91,2] = PR[GP1:90,2] + -0.045;
   1:L PR[91] R[100]mm/sec CNT100;
   1:  PR[GP1:91,1] = PR[GP1:90,1] + 60.498;
   1:  PR[GP1:91,2] = PR[GP1:90,2] + 0.578;
   1:L PR[91] R[100]mm/sec CNT100;
   1:  PR[GP1:91,1] = PR[GP1:90,1] + 58.251;
   1:  PR[GP1:91,2] = PR[GP1:90,2] + 12.699;
   1:L PR[91] R[100]mm/sec CNT100;
   1:  PR[GP1:91,1] = PR[GP1:90,1] + 58.119;
   1:  PR[GP1:91,2] = PR[GP1:90,2] + 13.142;
   1:L PR[91] R[100]mm/sec CNT100;
   1:  PR[GP1:91,1] = PR[GP1:90,1] + 57.898;
   1:  PR[GP1:91,2] = PR[GP1:90,2] + 13.570;
   1:L PR[91] R[100]mm/sec CNT100;
   1:  PR[GP1:91,1] = PR[GP1:90,1] + 51.201;
   1:  PR[GP1:91,2] = PR[GP1:90,2] + 24.694;
   1:L PR[91] R[100]mm/sec CNT100;
   1:  PR[GP1:91,1] = PR[GP1:90,1] + 51.104;
   1:  PR[GP1:91,2] = PR[GP1:90,2] + 24.820;
   1:L PR[91] R[100]mm/sec CNT100;
   1:  PR[GP1:91,1] = PR[GP1:90,1] + 50.989;
   1:  PR[GP1:91,2] = PR[GP1:90,2] + 24.922;
   1:L PR[91] R[100]mm/sec CNT100;
   1:  PR[GP1:91,1] = PR[GP1:90,1] + 45.743;
   1:  PR[GP1:91,2] = PR[GP1:90,2] + 29.157;
   1:L PR[91] R[100]mm/sec CNT100;
   1:  PR[GP1:91,1] = PR[GP1:90,1] + 40.633;
   1:  PR[GP1:91,2] = PR[GP1:90,2] + 33.379;
   1:L PR[91] R[100]mm/sec CNT100;
   1:  PR[GP1:91,1] = PR[GP1:90,1] + 40.291;
   1:  PR[GP1:91,2] = PR[GP1:90,2] + 33.650;
   1:L PR[91] R[100]mm/sec CNT100;
   1:  PR[GP1:91,1] = PR[GP1:90,1] + 28.387;
   1:  PR[GP1:91,2] = PR[GP1:90,2] + 38.040;
   1:L PR[91] R[100]mm/sec CNT100;
   1:  PR[GP1:91,1] = PR[GP1:90,1] + 26.779;
   1:  PR[GP1:91,2] = PR[GP1:90,2] + 38.568;
   1:L PR[91] R[100]mm/sec CNT100;
   1:  PR[GP1:91,1] = PR[GP1:90,1] + 15.109;
   1:  PR[GP1:91,2] = PR[GP1:90,2] + 38.779;
   1:L PR[91] R[100]mm/sec CNT100;
   1:  PR[GP1:91,1] = PR[GP1:90,1] + 12.160;
   1:  PR[GP1:91,2] = PR[GP1:90,2] + 38.673;
   1:L PR[91] R[100]mm/sec CNT100;
   1:  PR[GP1:91,1] = PR[GP1:90,1] + 3.417;
   1:  PR[GP1:91,2] = PR[GP1:90,2] + 35.971;
   1:L PR[91] R[100]mm/sec CNT100;
   1:  PR[GP1:91,1] = PR[GP1:90,1] + 2.127;
   1:  PR[GP1:91,2] = PR[GP1:90,2] + 35.554;
   1:L PR[91] R[100]mm/sec CNT100;
   1:  ! -- Layer/Ebene 127 -- !;
   1:  PR[91] = PR[90];
   1:  PR[GP1:91,1] = PR[GP1:90,1] + -1.886;
   1:  PR[GP1:91,2] = PR[GP1:90,2] + 35.745;
   1:  PR[GP1:91,3] = PR[GP1:90,3] + 77.775;
   1:L PR[91] R[100]mm/sec CNT100;
   1:  PR[GP1:91,1] = PR[GP1:90,1] + -11.652;
   1:  PR[GP1:91,2] = PR[GP1:90,2] + 38.763;
   1:L PR[91] R[100]mm/sec CNT100;
   1:  PR[GP1:91,1] = PR[GP1:90,1] + -14.937;
   1:  PR[GP1:91,2] = PR[GP1:90,2] + 38.881;
   1:L PR[91] R[100]mm/sec CNT100;
   1:  PR[GP1:91,1] = PR[GP1:90,1] + -26.307;
   1:  PR[GP1:91,2] = PR[GP1:90,2] + 38.673;
   1:L PR[91] R[100]mm/sec CNT100;
   1:  PR[GP1:91,1] = PR[GP1:90,1] + -28.244;
   1:  PR[GP1:91,2] = PR[GP1:90,2] + 38.038;
   1:L PR[91] R[100]mm/sec CNT100;
   1:  PR[GP1:91,1] = PR[GP1:90,1] + -39.858;
   1:  PR[GP1:91,2] = PR[GP1:90,2] + 33.752;
   1:L PR[91] R[100]mm/sec CNT100;
   1:  PR[GP1:91,1] = PR[GP1:90,1] + -40.481;
   1:  PR[GP1:91,2] = PR[GP1:90,2] + 33.258;
   1:L PR[91] R[100]mm/sec CNT100;
   1:  PR[GP1:91,1] = PR[GP1:90,1] + -48.998;
   1:  PR[GP1:91,2] = PR[GP1:90,2] + 26.229;
   1:L PR[91] R[100]mm/sec CNT100;
   1:  PR[GP1:91,1] = PR[GP1:90,1] + -50.692;
   1:  PR[GP1:91,2] = PR[GP1:90,2] + 24.857;
   1:L PR[91] R[100]mm/sec CNT100;
   1:  PR[GP1:91,1] = PR[GP1:90,1] + -57.726;
   1:  PR[GP1:91,2] = PR[GP1:90,2] + 13.116;
   1:L PR[91] R[100]mm/sec CNT100;
   1:  PR[GP1:91,1] = PR[GP1:90,1] + -57.799;
   1:  PR[GP1:91,2] = PR[GP1:90,2] + 12.866;
   1:L PR[91] R[100]mm/sec CNT100;
   1:  PR[GP1:91,1] = PR[GP1:90,1] + -57.833;
   1:  PR[GP1:91,2] = PR[GP1:90,2] + 12.501;
   1:L PR[91] R[100]mm/sec CNT100;
   1:  PR[GP1:91,1] = PR[GP1:90,1] + -60.156;
   1:  PR[GP1:91,2] = PR[GP1:90,2] + -0.100;
   1:L PR[91] R[100]mm/sec CNT100;
   1:  PR[GP1:91,1] = PR[GP1:90,1] + -60.115;
   1:  PR[GP1:91,2] = PR[GP1:90,2] + -0.546;
   1:L PR[91] R[100]mm/sec CNT100;
   1:  PR[GP1:91,1] = PR[GP1:90,1] + -57.806;
   1:  PR[GP1:91,2] = PR[GP1:90,2] + -12.987;
   1:L PR[91] R[100]mm/sec CNT100;
   1:  PR[GP1:91,1] = PR[GP1:90,1] + -57.718;
   1:  PR[GP1:91,2] = PR[GP1:90,2] + -13.284;
   1:L PR[91] R[100]mm/sec CNT100;
   1:  PR[GP1:91,1] = PR[GP1:90,1] + -57.573;
   1:  PR[GP1:91,2] = PR[GP1:90,2] + -13.569;
   1:L PR[91] R[100]mm/sec CNT100;
   1:  PR[GP1:91,1] = PR[GP1:90,1] + -50.713;
   1:  PR[GP1:91,2] = PR[GP1:90,2] + -24.983;
   1:L PR[91] R[100]mm/sec CNT100;
   1:  PR[GP1:91,1] = PR[GP1:90,1] + -50.680;
   1:  PR[GP1:91,2] = PR[GP1:90,2] + -25.018;
   1:L PR[91] R[100]mm/sec CNT100;
   1:  PR[GP1:91,1] = PR[GP1:90,1] + -48.999;
   1:  PR[GP1:91,2] = PR[GP1:90,2] + -26.373;
   1:L PR[91] R[100]mm/sec CNT100;
   1:  PR[GP1:91,1] = PR[GP1:90,1] + -40.471;
   1:  PR[GP1:91,2] = PR[GP1:90,2] + -33.408;
   1:L PR[91] R[100]mm/sec CNT100;
   1:  PR[GP1:91,1] = PR[GP1:90,1] + -39.847;
   1:  PR[GP1:91,2] = PR[GP1:90,2] + -33.902;
   1:L PR[91] R[100]mm/sec CNT100;
   1:  PR[GP1:91,1] = PR[GP1:90,1] + -28.230;
   1:  PR[GP1:91,2] = PR[GP1:90,2] + -38.184;
   1:L PR[91] R[100]mm/sec CNT100;
   1:  PR[GP1:91,1] = PR[GP1:90,1] + -26.292;
   1:  PR[GP1:91,2] = PR[GP1:90,2] + -38.820;
   1:L PR[91] R[100]mm/sec CNT100;
   1:  PR[GP1:91,1] = PR[GP1:90,1] + -14.921;
   1:  PR[GP1:91,2] = PR[GP1:90,2] + -39.022;
   1:L PR[91] R[100]mm/sec CNT100;
   1:  PR[GP1:91,1] = PR[GP1:90,1] + -11.637;
   1:  PR[GP1:91,2] = PR[GP1:90,2] + -38.905;
   1:L PR[91] R[100]mm/sec CNT100;
   1:  PR[GP1:91,1] = PR[GP1:90,1] + -1.888;
   1:  PR[GP1:91,2] = PR[GP1:90,2] + -35.870;
   1:L PR[91] R[100]mm/sec CNT100;
   1:  PR[GP1:91,1] = PR[GP1:90,1] + 2.098;
   1:  PR[GP1:91,2] = PR[GP1:90,2] + -35.868;
   1:L PR[91] R[100]mm/sec CNT100;
   1:  PR[GP1:91,1] = PR[GP1:90,1] + 11.848;
   1:  PR[GP1:91,2] = PR[GP1:90,2] + -38.904;
   1:L PR[91] R[100]mm/sec CNT100;
   1:  PR[GP1:91,1] = PR[GP1:90,1] + 15.132;
   1:  PR[GP1:91,2] = PR[GP1:90,2] + -39.021;
   1:L PR[91] R[100]mm/sec CNT100;
   1:  PR[GP1:91,1] = PR[GP1:90,1] + 26.503;
   1:  PR[GP1:91,2] = PR[GP1:90,2] + -38.820;
   1:L PR[91] R[100]mm/sec CNT100;
   1:  PR[GP1:91,1] = PR[GP1:90,1] + 28.442;
   1:  PR[GP1:91,2] = PR[GP1:90,2] + -38.184;
   1:L PR[91] R[100]mm/sec CNT100;
   1:  PR[GP1:91,1] = PR[GP1:90,1] + 40.058;
   1:  PR[GP1:91,2] = PR[GP1:90,2] + -33.905;
   1:L PR[91] R[100]mm/sec CNT100;
   1:  PR[GP1:91,1] = PR[GP1:90,1] + 40.683;
   1:  PR[GP1:91,2] = PR[GP1:90,2] + -33.411;
   1:L PR[91] R[100]mm/sec CNT100;
   1:  PR[GP1:91,1] = PR[GP1:90,1] + 49.211;
   1:  PR[GP1:91,2] = PR[GP1:90,2] + -26.369;
   1:L PR[91] R[100]mm/sec CNT100;
   1:  PR[GP1:91,1] = PR[GP1:90,1] + 50.920;
   1:  PR[GP1:91,2] = PR[GP1:90,2] + -24.986;
   1:L PR[91] R[100]mm/sec CNT100;
   1:  PR[GP1:91,1] = PR[GP1:90,1] + 57.936;
   1:  PR[GP1:91,2] = PR[GP1:90,2] + -13.285;
   1:L PR[91] R[100]mm/sec CNT100;
   1:  PR[GP1:91,1] = PR[GP1:90,1] + 58.009;
   1:  PR[GP1:91,2] = PR[GP1:90,2] + -13.040;
   1:L PR[91] R[100]mm/sec CNT100;
   1:  PR[GP1:91,1] = PR[GP1:90,1] + 58.044;
   1:  PR[GP1:91,2] = PR[GP1:90,2] + -12.666;
   1:L PR[91] R[100]mm/sec CNT100;
   1:  PR[GP1:91,1] = PR[GP1:90,1] + 60.369;
   1:  PR[GP1:91,2] = PR[GP1:90,2] + -0.045;
   1:L PR[91] R[100]mm/sec CNT100;
   1:  PR[GP1:91,1] = PR[GP1:90,1] + 60.326;
   1:  PR[GP1:91,2] = PR[GP1:90,2] + 0.417;
   1:L PR[91] R[100]mm/sec CNT100;
   1:  PR[GP1:91,1] = PR[GP1:90,1] + 58.019;
   1:  PR[GP1:91,2] = PR[GP1:90,2] + 12.866;
   1:L PR[91] R[100]mm/sec CNT100;
   1:  PR[GP1:91,1] = PR[GP1:90,1] + 57.932;
   1:  PR[GP1:91,2] = PR[GP1:90,2] + 13.156;
   1:L PR[91] R[100]mm/sec CNT100;
   1:  PR[GP1:91,1] = PR[GP1:90,1] + 57.786;
   1:  PR[GP1:91,2] = PR[GP1:90,2] + 13.440;
   1:L PR[91] R[100]mm/sec CNT100;
   1:  PR[GP1:91,1] = PR[GP1:90,1] + 50.904;
   1:  PR[GP1:91,2] = PR[GP1:90,2] + 24.852;
   1:L PR[91] R[100]mm/sec CNT100;
   1:  PR[GP1:91,1] = PR[GP1:90,1] + 49.211;
   1:  PR[GP1:91,2] = PR[GP1:90,2] + 26.224;
   1:L PR[91] R[100]mm/sec CNT100;
   1:  PR[GP1:91,1] = PR[GP1:90,1] + 40.693;
   1:  PR[GP1:91,2] = PR[GP1:90,2] + 33.262;
   1:L PR[91] R[100]mm/sec CNT100;
   1:  PR[GP1:91,1] = PR[GP1:90,1] + 40.069;
   1:  PR[GP1:91,2] = PR[GP1:90,2] + 33.755;
   1:L PR[91] R[100]mm/sec CNT100;
   1:  PR[GP1:91,1] = PR[GP1:90,1] + 28.455;
   1:  PR[GP1:91,2] = PR[GP1:90,2] + 38.038;
   1:L PR[91] R[100]mm/sec CNT100;
   1:  PR[GP1:91,1] = PR[GP1:90,1] + 26.518;
   1:  PR[GP1:91,2] = PR[GP1:90,2] + 38.674;
   1:L PR[91] R[100]mm/sec CNT100;
   1:  PR[GP1:91,1] = PR[GP1:90,1] + 15.148;
   1:  PR[GP1:91,2] = PR[GP1:90,2] + 38.880;
   1:L PR[91] R[100]mm/sec CNT100;
   1:  PR[GP1:91,1] = PR[GP1:90,1] + 11.863;
   1:  PR[GP1:91,2] = PR[GP1:90,2] + 38.762;
   1:L PR[91] R[100]mm/sec CNT100;
   1:  PR[GP1:91,1] = PR[GP1:90,1] + 2.094;
   1:  PR[GP1:91,2] = PR[GP1:90,2] + 35.743;
   1:L PR[91] R[100]mm/sec CNT100;
   1:  ! -- Layer/Ebene 128 -- !;
   1:  PR[91] = PR[90];
   1:  PR[GP1:91,1] = PR[GP1:90,1] + -1.860;
   1:  PR[GP1:91,2] = PR[GP1:90,2] + 35.918;
   1:  PR[GP1:91,3] = PR[GP1:90,3] + 78.385;
   1:L PR[91] R[100]mm/sec CNT100;
   1:  PR[GP1:91,1] = PR[GP1:90,1] + -11.354;
   1:  PR[GP1:91,2] = PR[GP1:90,2] + 38.851;
   1:L PR[91] R[100]mm/sec CNT100;
